	        //         IF #si_BinReleaseDistanceRight <= 0 THEN

	        //             #sx_Hold180 := TRUE;
	        //             #sx_ReleaseBinHoldRight := FALSE;
	        //             #sx_Hold170 := FALSE;
	        //             #sx_BinReleaseRight := FALSE;

	        //         END_IF;
	        //     END_IF;
	        // END_IF;

	    END_REGION


	    REGION Clearing sequence when workstation is deativated

	        #sF_TRIG_StationDeactivated(CLK := #ix_StationActive);



	        IF #sF_TRIG_StationDeactivated.Q THEN

	            #sx_Enable1X0In := TRUE;
	            #sx_Enable0X0In := TRUE;
	            #sx_Enable2X0In := TRUE;
	            #si_040DestinationA := 2;
	            #si_040DestinationB := 0;
	            #si_040DestinationC := 0;
	            #si_040DestinationD := 0;

	            #si_140DestinationA := 1;
	            #si_140DestinationB := 0;
	            #si_140DestinationC := 0;
	            #si_140DestinationD := 0;

	            #si_240DestinationA := 3;
	            #si_240DestinationB := 0;
	            #si_240DestinationC := 3;
	            #si_240DestinationD := 3;


	            #sx_Hold130 := FALSE;
	            #sx_Hold030 := FALSE;
	            #sx_Hold120 := FALSE;
	            #sx_Hold020 := FALSE;
	            #sx_Hold220 := FALSE;
	            #sx_Hold230 := FALSE;
	            #sx_Hold080 := FALSE;
	            #sx_Hold180 := FALSE;
	            #sx_StartClearing := TRUE;
	            #sx_NoOperationInProgress := FALSE;

	        END_IF;


	    END_REGION

	    REGION Finish operation

	        #sF_TRIG_ParcelArrived0X0(CLK := #iqUDT_WorkstationStatus."050".PEC_EoS.PEC);
	        #sF_TRIG_ParcelArrived1X0(CLK := #iqUDT_WorkstationStatus."150".PEC_EoS.PEC);
	        #sF_TRIG_ParcelArrived2X0(CLK := #iqUDT_WorkstationStatus."250".PEC_EoS.PEC);

	        // Check if operation if finished. If yes then set operation in progress bit
	        IF #si_SendTo0X0 AND #sF_TRIG_ParcelArrived0X0.Q OR #sFB_OperationTimeout.qx_DelayedSignal THEN

	            #si_SendTo0X0 := FALSE;

	        END_IF;


	        IF #si_SendTo1X0 AND #sF_TRIG_ParcelArrived1X0.Q OR #sFB_OperationTimeout.qx_DelayedSignal THEN

	            #si_SendTo1X0 := FALSE;

	        END_IF;

	        IF #si_SendTo2X0 AND #sF_TRIG_ParcelArrived2X0.Q OR #sFB_OperationTimeout.qx_DelayedSignal THEN

	            #si_SendTo2X0 := FALSE;

	        END_IF;


	        IF NOT #si_SendTo0X0 AND NOT #si_SendTo1X0 AND NOT #si_SendTo2X0 AND NOT #sx_StartClearing
	            AND #sUDT_Interface_040.ActualSpeed = 0
	            AND #sUDT_Interface_041.ActualSpeed = 0
	            AND #sUDT_Interface_140.ActualSpeed = 0
	            AND #sUDT_Interface_141.ActualSpeed = 0
	            AND #sUDT_Interface_240.ActualSpeed = 0
	            AND #sUDT_Interface_241.ActualSpeed = 0
	        THEN

	            #sx_NoOperationInProgress := TRUE;
	            #si_040DestinationA := 0;
	            #si_040DestinationB := 0;
	            #si_040DestinationC := 0;
	            #si_040DestinationD := 0;

	            #si_140DestinationA := 0;
	            #si_140DestinationB := 0;
	            #si_140DestinationC := 0;
	            #si_140DestinationD := 0;

	            #si_240DestinationA := 0;
	            #si_240DestinationB := 0;
	            #si_240DestinationC := 0;
	            #si_240DestinationD := 0;

	            #sx_Hold030 := FALSE;
	            #sx_Hold130 := FALSE;
	            #sx_Hold020 := FALSE;
	            #sx_Hold120 := FALSE;
	            #sx_Hold230 := FALSE;
	            #sx_Hold220 := FALSE;

	            #sx_Enable0X0In := FALSE;
	            #sx_Enable1X0In := FALSE;
	            #sx_Enable2X0In := FALSE;

	        END_IF;


	    END_REGION



	    REGION Workstation inicializaction

	        #sR_TRIG_InicializeWS(CLK := #ix_StationActive);

	        IF #sR_TRIG_InicializeWS.Q THEN

	            #sx_StartClearing := FALSE;
	            IF #iqUDT_WorkstationStatus."010".PEC_EoS.PEC THEN

	                #si_ReqestNewEmptyBin += 1;

	            END_IF;

	            IF #iqUDT_WorkstationStatus."020".PEC_EoS.PEC THEN

	                #si_ReqestNewEmptyBin += 1;

	            END_IF;

	            IF #iqUDT_WorkstationStatus."030".PEC_EoS.PEC THEN

	                #si_ReqestNewEmptyBin += 1;

	            END_IF;

	            IF #iqUDT_WorkstationStatus."110".PEC_EoS.PEC THEN

	                #si_ReqestNewPartialBin += 1;

	            END_IF;

	            IF #iqUDT_WorkstationStatus."120".PEC_EoS.PEC THEN

	                #si_ReqestNewPartialBin += 1;

	            END_IF;

	            IF #iqUDT_WorkstationStatus."130".PEC_EoS.PEC THEN

	                #si_ReqestNewPartialBin += 1;

	            END_IF;

	            #si_EmptyBinRequiredCounter0X0 := 2;
	            #si_EmptyBinRequiredCounter1X0 := 2;
	            #si_PartialyBinRequiredCounter0X0 := 1;
	            #si_PartialyBinRequiredCounter1X0 := 1;

	            REGION 050 Workposition inicialization
	                IF NOT #iqUDT_WorkstationStatus."050".PEC_EoS.PEC THEN
	                    IF #sa_TrackingArray_050[#iqUDT_Configuration."050".PEC_EoS.Distance / 10 - 2] > #iqUDT_Configuration.GlobalConfig.GINRangeStart
	                        AND #sa_TrackingArray_050[#iqUDT_Configuration."050".PEC_EoS.Distance / 10 - 2] < ((#iqUDT_Configuration.GlobalConfig.GINRangeStart + #iqUDT_Configuration.GlobalConfig.GINRangeEnd) / 2) THEN
	                        IF #si_EmptyBinRequiredCounter0X0 > 0 THEN
	                            #si_EmptyBinRequiredCounter0X0 -= 1;
	                        END_IF;
	                    ELSE

	                        IF #si_PartialyBinRequiredCounter0X0 > 0 THEN
	                            #si_PartialyBinRequiredCounter0X0 -= 1;
	                        ELSE
	                            IF #si_EmptyBinRequiredCounter0X0 > 0 THEN
	                                #si_EmptyBinRequiredCounter0X0 -= 1;
	                            END_IF;


	                        END_IF;

	                    END_IF;


	                END_IF;
	            END_REGION

	            REGION 060 Workposition inicialization
	                IF NOT #iqUDT_WorkstationStatus."060".PEC_EoS.PEC THEN
	                    IF #sa_TrackingArray_060[#iqUDT_Configuration."060".PEC_EoS.Distance / 10 - 2] > #iqUDT_Configuration.GlobalConfig.GINRangeStart
	                        AND #sa_TrackingArray_060[#iqUDT_Configuration."060".PEC_EoS.Distance / 10 - 2] < ((#iqUDT_Configuration.GlobalConfig.GINRangeStart + #iqUDT_Configuration.GlobalConfig.GINRangeEnd) / 2) THEN
	                        IF #si_EmptyBinRequiredCounter0X0 > 0 THEN
	                            #si_EmptyBinRequiredCounter0X0 -= 1;
	                        END_IF;
	                    ELSE

	                        IF #si_PartialyBinRequiredCounter0X0 > 0 THEN
	                            #si_PartialyBinRequiredCounter0X0 -= 1;
	                        ELSE
	                            IF #si_EmptyBinRequiredCounter0X0 > 0 THEN
	                                #si_EmptyBinRequiredCounter0X0 -= 1;
	                            END_IF;


	                        END_IF;

	                    END_IF;


	                END_IF;
	            END_REGION

	            REGION 070 Workposition inicialization
	                IF NOT #iqUDT_WorkstationStatus."070".PEC_EoS.PEC THEN
	                    IF #sa_TrackingArray_070[#iqUDT_Configuration."070".PEC_EoS.Distance / 10 - 2] > #iqUDT_Configuration.GlobalConfig.GINRangeStart
	                        AND #sa_TrackingArray_070[#iqUDT_Configuration."070".PEC_EoS.Distance / 10 - 2] < ((#iqUDT_Configuration.GlobalConfig.GINRangeStart + #iqUDT_Configuration.GlobalConfig.GINRangeEnd) / 2) THEN
	                        IF #si_EmptyBinRequiredCounter0X0 > 0 THEN
	                            #si_EmptyBinRequiredCounter0X0 -= 1;
	                        END_IF;
	                    ELSE

	                        IF #si_PartialyBinRequiredCounter0X0 > 0 THEN
	                            #si_PartialyBinRequiredCounter0X0 -= 1;
	                        ELSE
	                            IF #si_EmptyBinRequiredCounter0X0 > 0 THEN
	                                #si_EmptyBinRequiredCounter0X0 -= 1;
	                            END_IF;


	                        END_IF;

	                    END_IF;


	                END_IF;
	            END_REGION

	            REGION 150 Workposition inicialization
	                IF NOT #iqUDT_WorkstationStatus."150".PEC_EoS.PEC
	                THEN
	                    IF (#sa_TrackingArray_150[#iqUDT_Configuration."150".PEC_EoS.Distance / 10 / 10 - 2] > #iqUDT_Configuration.GlobalConfig.GINRangeStart
	                        AND #sa_TrackingArray_150[#iqUDT_Configuration."150".PEC_EoS.Distance / 10 - 2] < ((#iqUDT_Configuration.GlobalConfig.GINRangeStart + #iqUDT_Configuration.GlobalConfig.GINRangeEnd) / 2))
	                    THEN
	                        IF #si_EmptyBinRequiredCounter1X0 > 0 THEN
	                            #si_EmptyBinRequiredCounter1X0 -= 1;
	                        END_IF;
	                    ELSE

	                        IF #si_PartialyBinRequiredCounter1X0 > 0 THEN
	                            #si_PartialyBinRequiredCounter1X0 -= 1;
	                        ELSE
	                            IF #si_EmptyBinRequiredCounter1X0 > 0 THEN
	                                #si_EmptyBinRequiredCounter1X0 -= 1;
	                            END_IF;


	                        END_IF;

	                    END_IF;


	                END_IF;
	            END_REGION

	            REGION 160 Workposition inicialization
	                IF NOT #iqUDT_WorkstationStatus."160".PEC_EoS.PEC THEN
	                    IF #sa_TrackingArray_160[#iqUDT_Configuration."160".PEC_EoS.Distance / 10 - 2] > #iqUDT_Configuration.GlobalConfig.GINRangeStart
	                        AND #sa_TrackingArray_160[#iqUDT_Configuration."160".PEC_EoS.Distance / 10 - 2] < ((#iqUDT_Configuration.GlobalConfig.GINRangeStart + #iqUDT_Configuration.GlobalConfig.GINRangeEnd) / 2) THEN
	                        IF #si_EmptyBinRequiredCounter1X0 > 0 THEN
	                            #si_EmptyBinRequiredCounter1X0 -= 1;
	                        END_IF;
	                    ELSE

	                        IF #si_PartialyBinRequiredCounter1X0 > 0 THEN
	                            #si_PartialyBinRequiredCounter1X0 -= 1;
	                        ELSE
	                            IF #si_EmptyBinRequiredCounter1X0 > 0 THEN
	                                #si_EmptyBinRequiredCounter1X0 -= 1;
	                            END_IF;


	                        END_IF;

	                    END_IF;


	                END_IF;
	            END_REGION

	            REGION 170 Workposition inicialization
	                IF NOT #iqUDT_WorkstationStatus."170".PEC_EoS.PEC THEN
	                    IF #sa_TrackingArray_170[#iqUDT_Configuration."170".PEC_EoS.Distance / 10 - 2] > #iqUDT_Configuration.GlobalConfig.GINRangeStart
	                        AND #sa_TrackingArray_170[#iqUDT_Configuration."170".PEC_EoS.Distance / 10 - 2] < ((#iqUDT_Configuration.GlobalConfig.GINRangeStart + #iqUDT_Configuration.GlobalConfig.GINRangeEnd) / 2) THEN
	                        IF #si_EmptyBinRequiredCounter1X0 > 0 THEN
	                            #si_EmptyBinRequiredCounter1X0 -= 1;
	                        END_IF;
	                    ELSE

	                        IF #si_PartialyBinRequiredCounter1X0 > 0 THEN
	                            #si_PartialyBinRequiredCounter1X0 -= 1;
	                        ELSE
	                            IF #si_EmptyBinRequiredCounter1X0 > 0 THEN
	                                #si_EmptyBinRequiredCounter1X0 -= 1;
	                            END_IF;


	                        END_IF;

	                    END_IF;


	                END_IF;
	            END_REGION

	        END_IF;

	    END_REGION


	    REGION Request empty bin to buffer

	        IF #si_ReqestNewEmptyBin > 0 THEN

	            #ti_NumberOfBinInQueue := 0;
	            IF #iqUDT_EmptyBuffer.BufferState1.BinRequest THEN
	                #ti_NumberOfBinInQueue += 1;
	            END_IF;
	            IF #iqUDT_EmptyBuffer.BufferState2.BinRequest THEN
	                #ti_NumberOfBinInQueue += 1;
	            END_IF;
	            IF #iqUDT_EmptyBuffer.BufferState3.BinRequest THEN
	                #ti_NumberOfBinInQueue += 1;
	            END_IF;
	            IF NOT #iqUDT_WorkstationStatus."010".PEC_EoS.PEC THEN
	                #ti_NumberOfBinInQueue += 1;
	            END_IF;
	            IF NOT #iqUDT_WorkstationStatus."020".PEC_EoS.PEC THEN
	                #ti_NumberOfBinInQueue += 1;
	            END_IF;
	            IF NOT #iqUDT_WorkstationStatus."030".PEC_EoS.PEC THEN
	                #ti_NumberOfBinInQueue += 1;
	            END_IF;

	            IF #ti_NumberOfBinInQueue < 3 THEN

	                "FC_Fifo"(ic_Mode := 'S',
	                          qUDT_Status => #tUDT_FifoStatusEmpty,
	                          qx_Error => #tx_Error,
	                          qx_Warning => #tx_Warning,
	                          iqv_Data := #iqUDT_Configuration.GlobalConfig.DestinationEmpty,
	                          iqUDT_FifoHeader := #iqa_EmptyFifoHeader,
	                          iqv_DataBuffer := #iqa_EmptyFifoData);

	                IF NOT #tUDT_FifoStatusEmpty.FifoFull THEN

	                    "FC_Fifo"(ic_Mode := 'W',
	                              qUDT_Status => #tUDT_FifoStatusEmpty,
	                              qx_Error => #tx_Error,
	                              qx_Warning => #tx_Warning,
	                              iqv_Data := #iqUDT_Configuration.GlobalConfig.DestinationEmpty,
	                              iqUDT_FifoHeader := #iqa_EmptyFifoHeader,
	                              iqv_DataBuffer := #iqa_EmptyFifoData);

	                    IF NOT #iqUDT_EmptyBuffer.BufferState1.BinRequest THEN
	                        #iqUDT_EmptyBuffer.BufferState1.BinRequest := TRUE;
	                    ELSIF NOT #iqUDT_EmptyBuffer.BufferState2.BinRequest THEN
	                        #iqUDT_EmptyBuffer.BufferState2.BinRequest := TRUE;
	                    ELSE
	                        #iqUDT_EmptyBuffer.BufferState3.BinRequest := TRUE;
	                    END_IF;

	                    #si_ReqestNewEmptyBin -= 1;
	                    #iqUDT_EmptyBuffer.Destination := #iqUDT_Configuration.GlobalConfig.DestinationEmpty;
	                END_IF;



	            END_IF;

	        END_IF;


	    END_REGION

	    REGION Request partial bin to buffer

	        IF #si_ReqestNewPartialBin > 0 THEN

	            #ti_NumberOfBinInQueue := 0;
	            IF #iqUDT_PartialBuffer.BufferState1.BinRequest THEN
	                #ti_NumberOfBinInQueue += 1;
	            END_IF;
	            IF #iqUDT_PartialBuffer.BufferState2.BinRequest THEN
	                #ti_NumberOfBinInQueue += 1;
	            END_IF;
	            IF #iqUDT_PartialBuffer.BufferState3.BinRequest THEN
	                #ti_NumberOfBinInQueue += 1;
	            END_IF;
	            IF NOT #iqUDT_WorkstationStatus."110".PEC_EoS.PEC THEN
	                #ti_NumberOfBinInQueue += 1;
	            END_IF;
	            IF NOT #iqUDT_WorkstationStatus."120".PEC_EoS.PEC THEN
	                #ti_NumberOfBinInQueue += 1;
	            END_IF;
	            IF NOT #iqUDT_WorkstationStatus."130".PEC_EoS.PEC THEN
	                #ti_NumberOfBinInQueue += 1;
	            END_IF;

	            IF #ti_NumberOfBinInQueue < 3 THEN



	                "FC_Fifo"(ic_Mode := 'S',
	                          qUDT_Status => #tUDT_FifoStatusPartial,
	                          qx_Error => #tx_Error,
	                          qx_Warning => #tx_Warning,
	                          iqv_Data := #iqUDT_Configuration.GlobalConfig.DestinationPartialy,
	                          iqUDT_FifoHeader := #iqa_PartialFifoHeader,
	                          iqv_DataBuffer := #iqa_PartialFifoData);

	                IF NOT #tUDT_FifoStatusPartial.FifoFull THEN

	                    "FC_Fifo"(ic_Mode := 'W',
	                              qUDT_Status => #tUDT_FifoStatusPartial,
	                              qx_Error => #tx_Error,
	                              qx_Warning => #tx_Warning,
	                              iqv_Data := #iqUDT_Configuration.GlobalConfig.DestinationPartialy,
	                              iqUDT_FifoHeader := #iqa_PartialFifoHeader,
	                              iqv_DataBuffer := #iqa_PartialFifoData);

	                    IF NOT #iqUDT_PartialBuffer.BufferState1.BinRequest THEN
	                        #iqUDT_PartialBuffer.BufferState1.BinRequest := TRUE;
	                    ELSIF NOT #iqUDT_PartialBuffer.BufferState2.BinRequest THEN
	                        #iqUDT_PartialBuffer.BufferState2.BinRequest := TRUE;
	                    ELSE
	                        #iqUDT_PartialBuffer.BufferState3.BinRequest := TRUE;
	                    END_IF;

	                    #si_ReqestNewPartialBin -= 1;
	                    #iqUDT_PartialBuffer.Destination := #iqUDT_Configuration.GlobalConfig.DestinationPartialy;

	                END_IF;

	            END_IF;

	        END_IF;

	    END_REGION

	    REGION Ordered bin monitoring

	        IF "DB_Memory".OS_2sec THEN

	            IF #iqUDT_EmptyBuffer.BufferState1.BinSend THEN
	                #iqUDT_EmptyBuffer.BufferState1.WaintingTime += 2;

	                IF #iqUDT_EmptyBuffer.BufferState1.WaintingTime > #iqUDT_Configuration.GlobalConfig.BinOrderTimeout THEN

	                    #iqUDT_EmptyBuffer.BufferState1 := #iqUDT_EmptyBuffer.BufferState2;
	                    #iqUDT_EmptyBuffer.BufferState2 := #iqUDT_EmptyBuffer.BufferState3;

	                    #iqUDT_EmptyBuffer.BufferState3.BinSend := FALSE;
	                    #iqUDT_EmptyBuffer.BufferState3.BinRequest := FALSE;
	                    #iqUDT_EmptyBuffer.BufferState3.UpcomingBarcode := '';
	                    #iqUDT_EmptyBuffer.BufferState3.WaintingTime := 0;


	                    #ti_NumberOfBinInQueue := 0;
	                    IF #iqUDT_EmptyBuffer.BufferState1.BinRequest THEN
	                        #ti_NumberOfBinInQueue += 1;
	                    END_IF;
	                    IF #iqUDT_EmptyBuffer.BufferState2.BinRequest THEN
	                        #ti_NumberOfBinInQueue += 1;
	                    END_IF;
	                    IF NOT #iqUDT_WorkstationStatus."010".PEC_EoS.PEC THEN
	                        #ti_NumberOfBinInQueue += 1;
	                    END_IF;
	                    IF NOT #iqUDT_WorkstationStatus."020".PEC_EoS.PEC THEN
	                        #ti_NumberOfBinInQueue += 1;
	                    END_IF;
	                    IF NOT #iqUDT_WorkstationStatus."030".PEC_EoS.PEC THEN
	                        #ti_NumberOfBinInQueue += 1;
	                    END_IF;

	                    IF #ti_NumberOfBinInQueue < 3 THEN
	                        #si_ReqestNewEmptyBin += 1;
	                    END_IF;


	                END_IF;

	            END_IF;

	            IF #iqUDT_EmptyBuffer.BufferState2.BinSend THEN
	                #iqUDT_EmptyBuffer.BufferState2.WaintingTime += 2;

	                IF #iqUDT_EmptyBuffer.BufferState2.WaintingTime > #iqUDT_Configuration.GlobalConfig.BinOrderTimeout THEN

	                    #iqUDT_EmptyBuffer.BufferState2 := #iqUDT_EmptyBuffer.BufferState3;

	                    #iqUDT_EmptyBuffer.BufferState3.BinSend := FALSE;
	                    #iqUDT_EmptyBuffer.BufferState3.BinRequest := FALSE;
	                    #iqUDT_EmptyBuffer.BufferState3.UpcomingBarcode := '';
	                    #iqUDT_EmptyBuffer.BufferState3.WaintingTime := 0;

	                    #si_ReqestNewEmptyBin += 1;

	                END_IF;

	            END_IF;

	            IF #iqUDT_EmptyBuffer.BufferState3.BinSend THEN
	                #iqUDT_EmptyBuffer.BufferState3.WaintingTime += 2;

	                IF #iqUDT_EmptyBuffer.BufferState3.WaintingTime > #iqUDT_Configuration.GlobalConfig.BinOrderTimeout THEN

	                    #iqUDT_EmptyBuffer.BufferState3.BinSend := FALSE;
	                    #iqUDT_EmptyBuffer.BufferState3.BinRequest := FALSE;
	                    #iqUDT_EmptyBuffer.BufferState3.UpcomingBarcode := '';
	                    #iqUDT_EmptyBuffer.BufferState3.WaintingTime := 0;
	                    #si_ReqestNewEmptyBin += 1;

	                END_IF;

	            END_IF;

	            IF #iqUDT_PartialBuffer.BufferState1.BinSend THEN
	                #iqUDT_PartialBuffer.BufferState1.WaintingTime += 2;

	                IF #iqUDT_PartialBuffer.BufferState1.WaintingTime > #iqUDT_Configuration.GlobalConfig.BinOrderTimeout THEN

	                    #iqUDT_PartialBuffer.BufferState1 := #iqUDT_PartialBuffer.BufferState2;
	                    #iqUDT_PartialBuffer.BufferState2 := #iqUDT_PartialBuffer.BufferState3;
	                    #iqUDT_PartialBuffer.BufferState3.BinSend := FALSE;
	                    #iqUDT_PartialBuffer.BufferState3.BinRequest := FALSE;
	                    #iqUDT_PartialBuffer.BufferState3.UpcomingBarcode := '';
	                    #iqUDT_PartialBuffer.BufferState3.WaintingTime := 0;


	                    #ti_NumberOfBinInQueue := 0;
	                    IF #iqUDT_PartialBuffer.BufferState1.BinRequest THEN
	                        #ti_NumberOfBinInQueue += 1;
	                    END_IF;
	                    IF #iqUDT_PartialBuffer.BufferState2.BinRequest THEN
	                        #ti_NumberOfBinInQueue += 1;
	                    END_IF;
	                    IF NOT #iqUDT_WorkstationStatus."110".PEC_EoS.PEC THEN
	                        #ti_NumberOfBinInQueue += 1;
	                    END_IF;
	                    IF NOT #iqUDT_WorkstationStatus."120".PEC_EoS.PEC THEN
	                        #ti_NumberOfBinInQueue += 1;
	                    END_IF;
	                    IF NOT #iqUDT_WorkstationStatus."130".PEC_EoS.PEC THEN
	                        #ti_NumberOfBinInQueue += 1;
	                    END_IF;

	                    IF #ti_NumberOfBinInQueue < 3 THEN
	                        #si_ReqestNewPartialBin += 1;
	                    END_IF;

	                END_IF;

	            END_IF;


	            IF #iqUDT_PartialBuffer.BufferState2.BinSend THEN
	                #iqUDT_PartialBuffer.BufferState2.WaintingTime += 2;
	                IF #iqUDT_PartialBuffer.BufferState2.WaintingTime > #iqUDT_Configuration.GlobalConfig.BinOrderTimeout THEN

	                    #iqUDT_PartialBuffer.BufferState2 := #iqUDT_PartialBuffer.BufferState3;

	                    #iqUDT_PartialBuffer.BufferState3.BinSend := FALSE;
	                    #iqUDT_PartialBuffer.BufferState3.BinRequest := FALSE;
	                    #iqUDT_PartialBuffer.BufferState3.UpcomingBarcode := '';
	                    #iqUDT_PartialBuffer.BufferState3.WaintingTime := 0;

	                    #si_ReqestNewPartialBin += 1;

	                END_IF;

	            END_IF;

	            IF #iqUDT_PartialBuffer.BufferState3.BinSend THEN
	                #iqUDT_PartialBuffer.BufferState3.WaintingTime += 2;

	                IF #iqUDT_PartialBuffer.BufferState3.WaintingTime > #iqUDT_Configuration.GlobalConfig.BinOrderTimeout THEN

	                    #iqUDT_PartialBuffer.BufferState3.BinSend := FALSE;
	                    #iqUDT_PartialBuffer.BufferState3.BinRequest := FALSE;
	                    #iqUDT_PartialBuffer.BufferState3.UpcomingBarcode := '';
	                    #iqUDT_PartialBuffer.BufferState3.WaintingTime := 0;
	                    #si_ReqestNewPartialBin += 1;

	                END_IF;
	            END_IF;

	        END_IF;

	    END_REGION

	    REGION Ordered product confirmation

	        REGION Empty

	            #sR_TRIG_EmptyBinReceived(CLK := #sa_TrackingArray_010[#iqUDT_Configuration."010".PEC_EoS.Distance / 10 - 1] <> 0);

	            IF #sR_TRIG_EmptyBinReceived.Q THEN

	                IF #iqUDT_EmptyBuffer.BufferState1.BinSend AND "DB_GIN".GIN[#sa_TrackingArray_010[#iqUDT_Configuration."010".PEC_EoS.Distance / 10 - 1]].WES.Barcode = #iqUDT_EmptyBuffer.BufferState1.UpcomingBarcode THEN

	                    #iqUDT_EmptyBuffer.BufferState1 := #iqUDT_EmptyBuffer.BufferState2;
	                    #iqUDT_EmptyBuffer.BufferState2 := #iqUDT_EmptyBuffer.BufferState3;

	                    #iqUDT_EmptyBuffer.BufferState3.BinSend := FALSE;
	                    #iqUDT_EmptyBuffer.BufferState3.BinRequest := FALSE;
	                    #iqUDT_EmptyBuffer.BufferState3.UpcomingBarcode := '';
	                    #iqUDT_EmptyBuffer.BufferState3.WaintingTime := 0;
	                END_IF;


	                IF #iqUDT_EmptyBuffer.BufferState2.BinSend AND "DB_GIN".GIN[#sa_TrackingArray_010[#iqUDT_Configuration."010".PEC_EoS.Distance / 10 - 1]].WES.Barcode = #iqUDT_EmptyBuffer.BufferState2.UpcomingBarcode THEN

	                    #iqUDT_EmptyBuffer.BufferState2 := #iqUDT_EmptyBuffer.BufferState3;

	                    #iqUDT_EmptyBuffer.BufferState3.BinSend := FALSE;
	                    #iqUDT_EmptyBuffer.BufferState3.BinRequest := FALSE;
	                    #iqUDT_EmptyBuffer.BufferState3.UpcomingBarcode := '';
	                    #iqUDT_EmptyBuffer.BufferState3.WaintingTime := 0;
	                END_IF;


	                IF #iqUDT_EmptyBuffer.BufferState3.BinSend AND "DB_GIN".GIN[#sa_TrackingArray_010[#iqUDT_Configuration."010".PEC_EoS.Distance / 10 - 1]].WES.Barcode = #iqUDT_EmptyBuffer.BufferState3.UpcomingBarcode THEN

	                    #iqUDT_EmptyBuffer.BufferState3.BinSend := FALSE;
	                    #iqUDT_EmptyBuffer.BufferState3.BinRequest := FALSE;
	                    #iqUDT_EmptyBuffer.BufferState3.UpcomingBarcode := '';
	                    #iqUDT_EmptyBuffer.BufferState3.WaintingTime := 0;
	                END_IF;

	            END_IF;

	        END_REGION

	        REGION Partialy


	            #sR_TRIG_PartialBinReceived(CLK := #sa_TrackingArray_110[#iqUDT_Configuration."110".PEC_EoS.Distance / 10 - 1] <> 0);

	            IF #sR_TRIG_PartialBinReceived.Q THEN

	                IF #iqUDT_PartialBuffer.BufferState1.BinSend AND "DB_GIN".GIN[#sa_TrackingArray_110[#iqUDT_Configuration."110".PEC_EoS.Distance / 10 - 1]].WES.Barcode = #iqUDT_PartialBuffer.BufferState1.UpcomingBarcode THEN

	                    #iqUDT_PartialBuffer.BufferState1 := #iqUDT_PartialBuffer.BufferState2;
	                    #iqUDT_PartialBuffer.BufferState2 := #iqUDT_PartialBuffer.BufferState3;

	                    #iqUDT_PartialBuffer.BufferState3.BinSend := FALSE;
	                    #iqUDT_PartialBuffer.BufferState3.BinRequest := FALSE;
	                    #iqUDT_PartialBuffer.BufferState3.UpcomingBarcode := '';
	                    #iqUDT_PartialBuffer.BufferState3.WaintingTime := 0;
	                END_IF;


	                IF #iqUDT_PartialBuffer.BufferState2.BinSend AND "DB_GIN".GIN[#sa_TrackingArray_110[#iqUDT_Configuration."110".PEC_EoS.Distance / 10 - 1]].WES.Barcode = #iqUDT_PartialBuffer.BufferState2.UpcomingBarcode THEN

	                    #iqUDT_PartialBuffer.BufferState2 := #iqUDT_PartialBuffer.BufferState3;

	                    #iqUDT_PartialBuffer.BufferState3.BinSend := FALSE;
	                    #iqUDT_PartialBuffer.BufferState3.BinRequest := FALSE;
	                    #iqUDT_PartialBuffer.BufferState3.UpcomingBarcode := '';
	                    #iqUDT_PartialBuffer.BufferState3.WaintingTime := 0;
	                END_IF;


	                IF #iqUDT_PartialBuffer.BufferState3.BinSend AND "DB_GIN".GIN[#sa_TrackingArray_110[#iqUDT_Configuration."110".PEC_EoS.Distance / 10 - 1]].WES.Barcode = #iqUDT_PartialBuffer.BufferState3.UpcomingBarcode THEN

	                    #iqUDT_PartialBuffer.BufferState3.BinSend := FALSE;
	                    #iqUDT_PartialBuffer.BufferState3.BinRequest := FALSE;
	                    #iqUDT_PartialBuffer.BufferState3.UpcomingBarcode := '';
	                    #iqUDT_PartialBuffer.BufferState3.WaintingTime := 0;
	                END_IF;

	            END_IF;

	        END_REGION


	    END_REGION

	END_REGION

	REGION 010

	    REGION Change GIN range

	        #sR_TRIG_NewParcel010(CLK := #iqUDT_HandshakeUpstream010.GIN <> 0);

	        IF #sR_TRIG_NewParcel010.Q THEN

	            #si_LastGIN010 += 1;

	            IF #si_LastGIN010 < #iqUDT_Configuration.GlobalConfig.GINRangeStart
	                OR #si_LastGIN010 > ((#iqUDT_Configuration.GlobalConfig.GINRangeStart + #iqUDT_Configuration.GlobalConfig.GINRangeEnd) / 2)
	            THEN
	                #si_LastGIN010 := #iqUDT_Configuration.GlobalConfig.GINRangeStart;
	            END_IF;
	            #ts_Barcode := "DB_GIN".GIN[#iqUDT_HandshakeUpstream010.GIN].WES.Barcode;
	            #iqUDT_HandshakeUpstream010.GIN := #si_LastGIN010;
	            "DB_GIN".GIN[#iqUDT_HandshakeUpstream010.GIN] := "DB_GINDefault".GIN[#iqUDT_Configuration."010".PEC_EoS.DefaultGIN];
	            "DB_GIN".GIN[#iqUDT_HandshakeUpstream010.GIN].WES.Barcode := #ts_Barcode;
	        END_IF;

	    END_REGION

	    REGION Displacement
	        #sFB_Displacement010(#sUDT_Interface_010);
	    END_REGION

	    REGION Tracking

	        #sFB_Tracking_010(iUDT_ConveyorCommonConfiguration := #iqUDT_Configuration."010".Conveyor.Common,
	                          iqa_TrackingData := #sa_TrackingArray_010,
	                          iqUDT_ConveyorInterface := #sUDT_Interface_010,
	                          iqUDT_HandshakeUp := #iqUDT_HandshakeUpstream010,
	                          iqUDT_Handshake := #sUDT_Handshake_010);

	    END_REGION

	    REGION EoS

	        #sFB_PECUpdate_010(iUDT_PECUpdateConfiguration := #iqUDT_Configuration."010".PEC_EoS,
	                           iUDT_ConveyorCommonConfiguration := #iqUDT_Configuration."010".Conveyor.Common,
	                           ix_PEC := #iUDT_MotorInput010.AllSensorPortInputs.LeftSensor,
	                           ix_TeachingMode := FALSE,
	                           qUDT_Status => #iqUDT_WorkstationStatus."010".PEC_EoS,
	                           iqUDT_ConveyorInterface := #sUDT_Interface_010,
	                           iqUDT_UnknownGINRange := #iqUDT_UnknownGINRange,
	                           iqUDT_FifoHeader := "DB_FIFOLostGIN".Header,
	                           iqUDT_Statistics := #iqUDT_WorkstationStatistics."010".PEC_EoS,
	                           iqa_TrackingData := #sa_TrackingArray_010,
	                           iqa_FifoData := "DB_FIFOLostGIN".Data);

	    END_REGION

	    REGION Conveyor

	        #sFB_Conveyor_010(iUDT_ConveyorConfiguration := #iqUDT_Configuration."010".Conveyor,
	                          idi_PECEoSDistance := #iqUDT_Configuration."010".PEC_EoS.Distance,
	                          idi_PECBoSDistance := 0,
	                          ii_ExternalSpeed := 0,
	                          ix_SafetyOk := #ix_SafetyOk,
	                          ix_24vOk := #ix_24vOk,
	                          ix_400vOk := #ix_400vOk,
	                          ix_HardwareOk := TRUE,
	                          ix_PECEoS := #iqUDT_WorkstationStatus."010".PEC_EoS.PEC,
	                          ix_PECBoS := TRUE,
	                          ix_ReverseDirection := FALSE,
	                          ix_ExternalRequestDieBack := (#sUDT_Interface_020.ActualSpeed = 0 AND NOT #iqUDT_WorkstationStatus."010".PEC_EoS.PEC),
	                          ix_ExternalRequestHold := FALSE,
	                          ix_ResetEnergySave := FALSE,
	                          qUDT_HMIStatus => #iqUDT_WorkstationStatus."010".Conveyor,
	                          qUDT_Status => #iqUDT_WorkstationCommonStatus."010",
	                          iqUDT_EquipmentControl := #iqUDT_EquipmentControl,
	                          iqUDT_ConveyorCommand := #iqUDT_WorkstationCommands."010".Conveyor,
	                          iqUDT_ConveyorInterface := #sUDT_Interface_010,
	                          iqUDT_HandShakeUp := #iqUDT_HandshakeUpstream010,
	                          iqUDT_HandShake := #sUDT_Handshake_010,
	                          iqUDT_Statistics := #iqUDT_WorkstationStatistics."010".Conveyor);

	        // #iqUDT_HandshakeUpstream010.RTR := #iqUDT_HandshakeUpstream010.RTR AND #iqUDT_WorkstationStatus."010".PEC_EoS.PEC;

	    END_REGION

	    REGION MCO

	        #sFB_MCOConveyLinxAixController_010(iUDT_AixConfig := #iqUDT_Configuration."010".MCO_M01,
	                                            iUDT_AixInputsModule := #iUDT_MotorInput010,
	                                            ix_24vOk := #ix_24vOk,
	                                            ix_SimulationModeActive := "DB_Memory".Simulation,
	                                            ii_MotorPositionId := 1,
	                                            qUDT_HMIStatus => #iqUDT_WorkstationStatus."010".MCO_M01,
	                                            iqUDT_AixOutputsModule := #iqUDT_MotorOutput010,
	                                            iqUDT_ConveyorInterface := #sUDT_Interface_010,
	                                            iqUDT_MCOStatistics := #iqUDT_WorkstationStatistics."010".MCO_M01);
	    END_REGION

	END_REGION

	REGION 020

	    REGION Displacement
	        #sFB_Displacement020(#sUDT_Interface_020);
	    END_REGION

	    REGION Tracking

	        #sFB_Tracking_020(iUDT_ConveyorCommonConfiguration := #iqUDT_Configuration."020".Conveyor.Common,
	                          iqa_TrackingData := #sa_TrackingArray_020,
	                          iqUDT_ConveyorInterface := #sUDT_Interface_020,
	                          iqUDT_HandshakeUp := #sUDT_Handshake_010,
	                          iqUDT_Handshake := #sUDT_Handshake_020);

	    END_REGION

	    REGION EoS

	        #sFB_PECUpdate_020(iUDT_PECUpdateConfiguration := #iqUDT_Configuration."020".PEC_EoS,
	                           iUDT_ConveyorCommonConfiguration := #iqUDT_Configuration."020".Conveyor.Common,
	                           ix_PEC := #iUDT_MotorInput010.AllSensorPortInputs.RightSensor,
	                           ix_TeachingMode := FALSE,
	                           qUDT_Status => #iqUDT_WorkstationStatus."020".PEC_EoS,
	                           iqUDT_ConveyorInterface := #sUDT_Interface_020,
	                           iqUDT_UnknownGINRange := #iqUDT_UnknownGINRange,
	                           iqUDT_FifoHeader := "DB_FIFOLostGIN".Header,
	                           iqUDT_Statistics := #iqUDT_WorkstationStatistics."020".PEC_EoS,
	                           iqa_TrackingData := #sa_TrackingArray_020,
	                           iqa_FifoData := "DB_FIFOLostGIN".Data);




	    END_REGION

	    REGION Conveyor

	        #sFB_Conveyor_020(iUDT_ConveyorConfiguration := #iqUDT_Configuration."020".Conveyor,
	                          idi_PECEoSDistance := #iqUDT_Configuration."020".PEC_EoS.Distance,
	                          idi_PECBoSDistance := 0,
	                          ii_ExternalSpeed := 0,
	                          ix_SafetyOk := #ix_SafetyOk,
	                          ix_24vOk := #ix_24vOk,
	                          ix_400vOk := #ix_400vOk,
	                          ix_HardwareOk := TRUE,
	                          ix_PECEoS := #iqUDT_WorkstationStatus."020".PEC_EoS.PEC,
	                          ix_PECBoS := TRUE,
	                          ix_ReverseDirection := FALSE,
	                          ix_ExternalRequestDieBack := #sx_Hold020 OR (#sUDT_Interface_030.ActualSpeed = 0 AND NOT #iqUDT_WorkstationStatus."020".PEC_EoS.PEC),
	                          ix_ExternalRequestHold := FALSE,
	                          ix_ResetEnergySave := FALSE,
	                          qUDT_HMIStatus => #iqUDT_WorkstationStatus."020".Conveyor,
	                          qUDT_Status => #iqUDT_WorkstationCommonStatus."020",
	                          iqUDT_EquipmentControl := #iqUDT_EquipmentControl,
	                          iqUDT_ConveyorCommand := #iqUDT_WorkstationCommands."020".Conveyor,
	                          iqUDT_ConveyorInterface := #sUDT_Interface_020,
	                          iqUDT_HandShakeUp := #sUDT_Handshake_010,
	                          iqUDT_HandShake := #sUDT_Handshake_020,
	                          iqUDT_Statistics := #iqUDT_WorkstationStatistics."020".Conveyor);

	    END_REGION

	    REGION MCO

	        #sFB_MCOConveyLinxAixController_020(iUDT_AixConfig := #iqUDT_Configuration."020".MCO_M01,
	                                            iUDT_AixInputsModule := #iUDT_MotorInput010,
	                                            ix_24vOk := #ix_24vOk,
	                                            ix_SimulationModeActive := "DB_Memory".Simulation,
	                                            ii_MotorPositionId := 2,
	                                            qUDT_HMIStatus => #iqUDT_WorkstationStatus."020".MCO_M01,
	                                            iqUDT_AixOutputsModule := #iqUDT_MotorOutput010,
	                                            iqUDT_ConveyorInterface := #sUDT_Interface_020,
	                                            iqUDT_MCOStatistics := #iqUDT_WorkstationStatistics."020".MCO_M01);
	    END_REGION

	END_REGION

	REGION 030

	    REGION Displacement
	        #sFB_Displacement030(#sUDT_Interface_030);
	    END_REGION

	    REGION Tracking

	        #sFB_Tracking_030(iUDT_ConveyorCommonConfiguration := #iqUDT_Configuration."030".Conveyor.Common,
	                          iqa_TrackingData := #sa_TrackingArray_030,
	                          iqUDT_ConveyorInterface := #sUDT_Interface_030,
	                          iqUDT_HandshakeUp := #sUDT_Handshake_020,
	                          iqUDT_Handshake := #sUDT_Handshake_030);

	    END_REGION

	    REGION EoS

	        #sFB_PECUpdate_030(iUDT_PECUpdateConfiguration := #iqUDT_Configuration."030".PEC_EoS,
	                           iUDT_ConveyorCommonConfiguration := #iqUDT_Configuration."030".Conveyor.Common,
	                           ix_PEC := #iUDT_MotorInput030.AllSensorPortInputs.LeftSensor,
	                           ix_TeachingMode := FALSE,
	                           qUDT_Status => #iqUDT_WorkstationStatus."030".PEC_EoS,
	                           iqUDT_ConveyorInterface := #sUDT_Interface_030,
	                           iqUDT_UnknownGINRange := #iqUDT_UnknownGINRange,
	                           iqUDT_FifoHeader := "DB_FIFOLostGIN".Header,
	                           iqUDT_Statistics := #iqUDT_WorkstationStatistics."030".PEC_EoS,
	                           iqa_TrackingData := #sa_TrackingArray_030,
	                           iqa_FifoData := "DB_FIFOLostGIN".Data);




	    END_REGION

	    REGION Conveyor

	        #sUDT_Handshake_030.RTR := #sUDT_Handshake_030.RTR AND NOT #sx_Hold030 OR #iqUDT_WorkstationStatus."030".PEC_EoS.PEC;


	        #sFB_Conveyor_030(iUDT_ConveyorConfiguration := #iqUDT_Configuration."030".Conveyor,
	                          idi_PECEoSDistance := #iqUDT_Configuration."030".PEC_EoS.Distance,
	                          idi_PECBoSDistance := 0,
	                          ii_ExternalSpeed := 0,
	                          ix_SafetyOk := #ix_SafetyOk,
	                          ix_24vOk := #ix_24vOk,
	                          ix_400vOk := #ix_400vOk,
	                          ix_HardwareOk := TRUE,
	                          ix_PECEoS := #iqUDT_WorkstationStatus."030".PEC_EoS.PEC,
	                          ix_PECBoS := TRUE,
	                          ix_ReverseDirection := FALSE,
	                          ix_ExternalRequestDieBack := FALSE,
	                          ix_ExternalRequestHold := #sx_Hold030,
	                          ix_ResetEnergySave := FALSE,
	                          qUDT_HMIStatus => #iqUDT_WorkstationStatus."030".Conveyor,
	                          qUDT_Status => #iqUDT_WorkstationCommonStatus."030",
	                          iqUDT_EquipmentControl := #iqUDT_EquipmentControl,
	                          iqUDT_ConveyorCommand := #iqUDT_WorkstationCommands."030".Conveyor,
	                          iqUDT_ConveyorInterface := #sUDT_Interface_030,
	                          iqUDT_HandShakeUp := #sUDT_Handshake_020,
	                          iqUDT_HandShake := #sUDT_Handshake_030,
	                          iqUDT_Statistics := #iqUDT_WorkstationStatistics."030".Conveyor);

	    END_REGION

	    REGION MCO

	        #sFB_MCOConveyLinxAixController_030(iUDT_AixConfig := #iqUDT_Configuration."030".MCO_M01,
	                                            iUDT_AixInputsModule := #iUDT_MotorInput030,
	                                            ix_24vOk := #ix_24vOk,
	                                            ix_SimulationModeActive := "DB_Memory".Simulation,
	                                            ii_MotorPositionId := 1,
	                                            qUDT_HMIStatus => #iqUDT_WorkstationStatus."030".MCO_M01,
	                                            iqUDT_AixOutputsModule := #iqUDT_MotorOutput030,
	                                            iqUDT_ConveyorInterface := #sUDT_Interface_030,
	                                            iqUDT_MCOStatistics := #iqUDT_WorkstationStatistics."030".MCO_M01);
	    END_REGION

	END_REGION

	REGION 040

	    REGION Displacement
	        #sFB_Displacement040(#sUDT_Interface_040);
	    END_REGION

	    REGION MCO

	        #sFB_MCOConveyLinxAixController_040(iUDT_AixConfig := #iqUDT_Configuration."040".MCO_M01,
	                                            iUDT_AixInputsModule := #iUDT_MotorInput040,
	                                            ii_PositionSetpoint := #iqUDT_RATPositioning040.Lower.EndPosition,
	                                            ix_24vOk := #ix_24vOk,
	                                            ix_SimulationModeActive := "DB_Memory".Simulation,
	                                            ii_MotorPositionId := 1,
	                                            ix_StartPositioning := #iqUDT_RATPositioning040.Lower.Start,
	                                            ix_ResetPosition := #iqUDT_RATPositioning040.Lower.ResetPosition,
	                                            qUDT_HMIStatus => #iqUDT_WorkstationStatus."040".MCO_M01,
	                                            qx_Positioned => #iqUDT_RATPositioning040.Lower.Done,
	                                            iqUDT_AixOutputsModule := #iqUDT_MotorOutput040,
	                                            iqUDT_ConveyorInterface := #sUDT_Interface_040,
	                                            iqUDT_MCOStatistics := #iqUDT_WorkstationStatistics."040".MCO_M01);
	    END_REGION

	    REGION BladeStopEoS

	        IF #iqUDT_Configuration.GlobalConfig.LeftStationAvailable THEN

	            #sFB_BladeStopEoS_040(iUDT_Configuration := #iqUDT_Configuration."040".BladeStopEoS,
	                                  ix_IsOpened := #ix_BladeStopisUp040,
	                                  ix_IsClosed := #ix_BladeStopisDown040,
	                                  ix_AirPressureOk := TRUE,
	                                  qx_Open => #qx_BladeStopControl040,
	                                  qUDT_HMIStatus => #iqUDT_WorkstationStatus."040".BladeStopEoS,
	                                  qUDT_Statistics => #iqUDT_WorkstationStatistics."040".BladeStopEoS,
	                                  iqUDT_EquipmentControl := #iqUDT_EquipmentControl,
	                                  iqUDT_HMICommand := #iqUDT_WorkstationCommands."040".BladeStopEoS,
	                                  iqUDT_Interface := #sUDT_Interface_040_BladeStopEoS);
	        END_IF;

	    END_REGION

	END_REGION

	REGION 041

	    REGION Displacement
	        #sFB_Displacement041(#sUDT_Interface_041);
	    END_REGION

	    REGION RAT

	        #iqUDT_Configuration."041".RightAngledTransfer.BladeStopEoS := #iqUDT_Configuration.GlobalConfig.LeftStationAvailable;

	        #sFB_RightAngledTransfer_041(iUDT_Configuration := #iqUDT_Configuration."041".RightAngledTransfer,
	                                     iUDT_LowerConveyorConfiguration := #iqUDT_Configuration."040".Conveyor,
	                                     iUDT_UpperConveyorConfiguration := #iqUDT_Configuration."041".Conveyor,
	                                     iUDT_PECConfiguration := #iqUDT_Configuration."040".PEC_EoS,
	                                     ii_DestinationA := #si_040DestinationA,
	                                     ii_DestinationB := #si_040DestinationB,
	                                     ii_DestinationC := #si_040DestinationC,
	                                     ii_DestinationD := #si_040DestinationD,
	                                     ix_HardwareOk := TRUE,
	                                     ix_400vOk := #ix_400vOk,
	                                     ix_24vOk := #ix_24vOk,
	                                     ix_SafetyOk := #ix_SafetyOk,
	                                     ix_AirPressureOk := #ix_AirPressureOk,
	                                     ix_SectionIsDown := #ix_SectionisDown041,
	                                     ix_SectionIsUp := #ix_SectionisUp041,
	                                     ix_ConveyorAAuto := #iqUDT_WorkstationCommonStatus."030".AutoON,
	                                     ix_ConveyorBAuto := #iqUDT_WorkstationCommonStatus."050".AutoON,
	                                     ix_ConveyorCAuto := FALSE,
	                                     ix_ConveyorDAuto := #iqUDT_WorkstationCommonStatus."241".AutoON,
	                                     ix_PEC := #iUDT_MotorInput040.AllSensorPortInputs.LeftSensor,
	                                     ix_ExternalReceiveRequestA := NOT #iqUDT_WorkstationStatus."030".PEC_EoS.PEC AND #sx_Enable0X0In,
	                                     ix_ExternalReceiveRequestB := false,
	                                     ix_ExternalReceiveRequestC := false,
	                                     ix_ExternalReceiveRequestD := #sFB_RightAngledTransfer_241.qx_ExternalSendRequestD,
	                                     ix_PECInfeedA := #iqUDT_WorkstationStatus."030".PEC_EoS.PEC,
	                                     ix_PECInfeedD := #iqUDT_WorkstationStatus."240".PEC_EoS.PEC,
	                                     qUDT_HMIRATStatus => #iqUDT_WorkstationStatus."041".RightAngledTransfer,
	                                     qUDT_HMIConveyorStatus => #iqUDT_WorkstationStatus."040".Conveyor,
	                                     qUDT_HMIPECStatus => #iqUDT_WorkstationStatus."040".PEC_EoS,
	                                     qUDT_RATStatus => #iqUDT_WorkstationCommonStatus."041",
	                                     qUDT_ConveyorStatus => #iqUDT_WorkstationCommonStatus."040",
	                                     qx_PopupControl => #qx_PopupControl041,
	                                     iqUDT_EquipmentControl := #iqUDT_EquipmentControl,
	                                     iqUDT_RATCommand := #iqUDT_WorkstationCommands."041".RightAngledTransfer,
	                                     iqUDT_ConveyorCommand := #iqUDT_WorkstationCommands."040".Conveyor,
	                                     iqUDT_RATStatistics := #iqUDT_WorkstationStatistics."041".RightAngledTransfer,
	                                     iqUDT_ConveyorStatistics := #iqUDT_WorkstationStatistics."040".Conveyor,
	                                     iqUDT_PECStatistics := #iqUDT_WorkstationStatistics."040".PEC_EoS,
	                                     iqUDT_HandShakeConveyorA := #sUDT_Handshake_030,
	                                     iqUDT_HandShakeConveyorB := #sUDT_Handshake_040,
	                                     iqUDT_HandShakeConveyorC := #sUDT_HandshakeUp_041,
	                                     iqUDT_HandShakeConveyorD := #sUDT_Handshake_041,
	                                     iqUDT_LowerConveyorInterface := #sUDT_Interface_040,
	                                     iqUDT_UpperConveyorInterface := #sUDT_Interface_041,
	                                     iqUDT_RATPositioning := #iqUDT_RATPositioning040,
	                                     iqUDT_BladeStopEoSInterface := #sUDT_Interface_040_BladeStopEoS,
	                                     iqUDT_BladeStopBoSInterface := #tUDT_DummyBladeStop);

	    END_REGION

	    REGION MCO

	        #sFB_MCOConveyLinxAixController_041(iUDT_AixConfig := #iqUDT_Configuration."041".MCO_M01,
	                                            iUDT_AixInputsModule := #iUDT_MotorInput040,
	                                            ii_PositionSetpoint := #iqUDT_RATPositioning040.Upper.EndPosition,
	                                            ix_24vOk := #ix_24vOk,
	                                            ix_SimulationModeActive := "DB_Memory".Simulation,
	                                            ii_MotorPositionId := 2,
	                                            ix_StartPositioning := #iqUDT_RATPositioning040.Upper.Start,
	                                            qUDT_HMIStatus => #iqUDT_WorkstationStatus."041".MCO_M01,
	                                            qx_Positioned => #iqUDT_RATPositioning040.Upper.Done,
	                                            iqUDT_AixOutputsModule := #iqUDT_MotorOutput040,
	                                            iqUDT_ConveyorInterface := #sUDT_Interface_041,
	                                            iqUDT_MCOStatistics := #iqUDT_WorkstationStatistics."041".MCO_M01);
	    END_REGION

	END_REGION

	IF #iqUDT_Configuration.GlobalConfig.LeftStationAvailable THEN

	    REGION 050

	        REGION Displacement
	            #sFB_Displacement050(#sUDT_Interface_050);
	        END_REGION

	        REGION Tracking

	            #sFB_Tracking_050(iUDT_ConveyorCommonConfiguration := #iqUDT_Configuration."050".Conveyor.Common,
	                              iqa_TrackingData := #sa_TrackingArray_050,
	                              iqUDT_ConveyorInterface := #sUDT_Interface_050,
	                              iqUDT_HandshakeUp := #sUDT_Handshake_040,
	                              iqUDT_Handshake := #sUDT_Handshake_050);

	        END_REGION

	        REGION EoS

	            #sFB_PECUpdate_050(iUDT_PECUpdateConfiguration := #iqUDT_Configuration."050".PEC_EoS,
	                               iUDT_ConveyorCommonConfiguration := #iqUDT_Configuration."050".Conveyor.Common,
	                               ix_PEC := NOT #iUDT_MotorInput050.AllSensorPortInputs.LeftSensor,
	                               ix_TeachingMode := FALSE,
	                               qUDT_Status => #iqUDT_WorkstationStatus."050".PEC_EoS,
	                               iqUDT_ConveyorInterface := #sUDT_Interface_050,
	                               iqUDT_UnknownGINRange := #iqUDT_UnknownGINRange,
	                               iqUDT_FifoHeader := "DB_FIFOLostGIN".Header,
	                               iqUDT_Statistics := #iqUDT_WorkstationStatistics."050".PEC_EoS,
	                               iqa_TrackingData := #sa_TrackingArray_050,
	                               iqa_FifoData := "DB_FIFOLostGIN".Data);

	        END_REGION

	        REGION Conveyor

	            //#sUDT_Handshake_050.RTR := TRUE;

	            #sUDT_Handshake_050.RTR := (#iqUDT_WorkstationStatus."060".PEC_EoS.PEC AND #sUDT_Interface_060.ActualSpeed <> 0)
	            OR (#iqUDT_WorkstationStatus."050".PEC_EoS.PEC);

	            #sFB_Conveyor_050(iUDT_ConveyorConfiguration := #iqUDT_Configuration."050".Conveyor,
	                              idi_PECEoSDistance := #iqUDT_Configuration."050".PEC_EoS.Distance,
	                              idi_PECBoSDistance := 0,
	                              ii_ExternalSpeed := 0,
	                              ix_SafetyOk := #ix_SafetyOk,
	                              ix_24vOk := #ix_24vOk,
	                              ix_400vOk := #ix_400vOk,
	                              ix_HardwareOk := TRUE,
	                              ix_PECEoS := #iqUDT_WorkstationStatus."050".PEC_EoS.PEC,
	                              ix_PECBoS := TRUE,
	                              ix_ReverseDirection := FALSE,
	                              ix_ExternalRequestDieBack := FALSE,
	                              ix_ExternalRequestHold := #sx_ReleaseBinHoldLeft,//NOT #tx_Enable,
	                              ix_ResetEnergySave := FALSE,
	                              qUDT_HMIStatus => #iqUDT_WorkstationStatus."050".Conveyor,
	                              qUDT_Status => #iqUDT_WorkstationCommonStatus."050",
	                              iqUDT_EquipmentControl := #iqUDT_EquipmentControl,
	                              iqUDT_ConveyorCommand := #iqUDT_WorkstationCommands."050".Conveyor,
	                              iqUDT_ConveyorInterface := #sUDT_Interface_050,
	                              iqUDT_HandShakeUp := #sUDT_Handshake_040,
	                              iqUDT_HandShake := #sUDT_Handshake_050,
	                              iqUDT_Statistics := #iqUDT_WorkstationStatistics."050".Conveyor);

	        END_REGION

	        REGION MCO

	            #sFB_MCOConveyLinxAixController_050(iUDT_AixConfig := #iqUDT_Configuration."050".MCO_M01,
	                                                iUDT_AixInputsModule := #iUDT_MotorInput050,
	                                                ix_24vOk := #ix_24vOk,
	                                                ix_SimulationModeActive := "DB_Memory".Simulation,
	                                                ii_MotorPositionId := 1,
	                                                qUDT_HMIStatus => #iqUDT_WorkstationStatus."050".MCO_M01,
	                                                iqUDT_AixOutputsModule := #iqUDT_MotorOutput050,
	                                                iqUDT_ConveyorInterface := #sUDT_Interface_050,
	                                                iqUDT_MCOStatistics := #iqUDT_WorkstationStatistics."050".MCO_M01);
	        END_REGION

	    END_REGION

	    REGION 060

	        REGION Displacement
	            #sFB_Displacement060(#sUDT_Interface_060);
	        END_REGION

	        REGION Tracking

	            #sFB_Tracking_060(iUDT_ConveyorCommonConfiguration := #iqUDT_Configuration."060".Conveyor.Common,
	                              iqa_TrackingData := #sa_TrackingArray_060,
	                              iqUDT_ConveyorInterface := #sUDT_Interface_060,
	                              iqUDT_HandshakeUp := #sUDT_Handshake_050,
	                              iqUDT_Handshake := #sUDT_Handshake_060);

	        END_REGION

	        REGION EoS

	            #sFB_PECUpdate_060(iUDT_PECUpdateConfiguration := #iqUDT_Configuration."060".PEC_EoS,
	                               iUDT_ConveyorCommonConfiguration := #iqUDT_Configuration."060".Conveyor.Common,
	                               ix_PEC := NOT #iUDT_MotorInput050.AllSensorPortInputs.RightSensor,
	                               ix_TeachingMode := FALSE,
	                               qUDT_Status => #iqUDT_WorkstationStatus."060".PEC_EoS,
	                               iqUDT_ConveyorInterface := #sUDT_Interface_060,
	                               iqUDT_UnknownGINRange := #iqUDT_UnknownGINRange,
	                               iqUDT_FifoHeader := "DB_FIFOLostGIN".Header,
	                               iqUDT_Statistics := #iqUDT_WorkstationStatistics."060".PEC_EoS,
	                               iqa_TrackingData := #sa_TrackingArray_060,
	                               iqa_FifoData := "DB_FIFOLostGIN".Data);

	        END_REGION

	        REGION Conveyor

	            // #sUDT_Handshake_060.RTR := TRUE;

	            #sUDT_Handshake_060.RTR := (#iqUDT_WorkstationStatus."070".PEC_EoS.PEC AND #sUDT_Interface_070.ActualSpeed <> 0)
	            OR (#iqUDT_WorkstationStatus."060".PEC_EoS.PEC);

	            #sFB_Conveyor_060(iUDT_ConveyorConfiguration := #iqUDT_Configuration."060".Conveyor,
	                              idi_PECEoSDistance := #iqUDT_Configuration."060".PEC_EoS.Distance,
	                              idi_PECBoSDistance := 0,
	                              ii_ExternalSpeed := 0,
	                              ix_SafetyOk := #ix_SafetyOk,
	                              ix_24vOk := #ix_24vOk,
	                              ix_400vOk := #ix_400vOk,
	                              ix_HardwareOk := TRUE,
	                              ix_PECEoS := #iqUDT_WorkstationStatus."060".PEC_EoS.PEC,
	                              ix_PECBoS := TRUE,
	                              ix_ReverseDirection := FALSE,
	                              ix_ExternalRequestDieBack := FALSE,
	                              ix_ExternalRequestHold := #sx_ReleaseBinHoldLeft,//NOT #tx_Enable,//(NOT #iqUDT_WorkstationStatus."035"."036".PEC_EoS.PEC AND NOT #iqUDT_WorkstationStatus."030"."031".PEC_EoS.PEC) OR (#sUDT_Interface_036.ActualSpeed = 0 AND #iqUDT_WorkstationStatus."030"."031".PEC_EoS.PEC),
	                              ix_ResetEnergySave := FALSE,
	                              qUDT_HMIStatus => #iqUDT_WorkstationStatus."060".Conveyor,
	                              qUDT_Status => #iqUDT_WorkstationCommonStatus."060",
	                              iqUDT_EquipmentControl := #iqUDT_EquipmentControl,
	                              iqUDT_ConveyorCommand := #iqUDT_WorkstationCommands."060".Conveyor,
	                              iqUDT_ConveyorInterface := #sUDT_Interface_060,
	                              iqUDT_HandShakeUp := #sUDT_Handshake_050,
	                              iqUDT_HandShake := #sUDT_Handshake_060,
	                              iqUDT_Statistics := #iqUDT_WorkstationStatistics."060".Conveyor);

	        END_REGION

	        REGION MCO

	            #sFB_MCOConveyLinxAixController_060(iUDT_AixConfig := #iqUDT_Configuration."060".MCO_M01,
	                                                iUDT_AixInputsModule := #iUDT_MotorInput050,
	                                                ix_24vOk := #ix_24vOk,
	                                                ix_SimulationModeActive := "DB_Memory".Simulation,
	                                                ii_MotorPositionId := 2,
	                                                qUDT_HMIStatus => #iqUDT_WorkstationStatus."060".MCO_M01,
	                                                iqUDT_AixOutputsModule := #iqUDT_MotorOutput050,
	                                                iqUDT_ConveyorInterface := #sUDT_Interface_060,
	                                                iqUDT_MCOStatistics := #iqUDT_WorkstationStatistics."060".MCO_M01);
	        END_REGION

	    END_REGION

	    REGION 070

	        REGION Displacement
	            #sFB_Displacement070(#sUDT_Interface_070);
	        END_REGION

	        REGION Tracking

	            #sFB_Tracking_070(iUDT_ConveyorCommonConfiguration := #iqUDT_Configuration."070".Conveyor.Common,
	                              iqa_TrackingData := #sa_TrackingArray_070,
	                              iqUDT_ConveyorInterface := #sUDT_Interface_070,
	                              iqUDT_HandshakeUp := #sUDT_Handshake_060,
	                              iqUDT_Handshake := #sUDT_Handshake_070);

	        END_REGION

	        REGION EoS

	            #sFB_PECUpdate_070(iUDT_PECUpdateConfiguration := #iqUDT_Configuration."070".PEC_EoS,
	                               iUDT_ConveyorCommonConfiguration := #iqUDT_Configuration."070".Conveyor.Common,
	                               ix_PEC := NOT #iUDT_MotorInput070.AllSensorPortInputs.LeftSensor,
	                               ix_TeachingMode := FALSE,
	                               qUDT_Status => #iqUDT_WorkstationStatus."070".PEC_EoS,
	                               iqUDT_ConveyorInterface := #sUDT_Interface_070,
	                               iqUDT_UnknownGINRange := #iqUDT_UnknownGINRange,
	                               iqUDT_FifoHeader := "DB_FIFOLostGIN".Header,
	                               iqUDT_Statistics := #iqUDT_WorkstationStatistics."070".PEC_EoS,
	                               iqa_TrackingData := #sa_TrackingArray_070,
	                               iqa_FifoData := "DB_FIFOLostGIN".Data);

	        END_REGION

	        REGION Conveyor

	            #sUDT_Handshake_070.RTR := #iqUDT_WorkstationStatus."070".PEC_EoS.PEC;

	            #sFB_Conveyor_070(iUDT_ConveyorConfiguration := #iqUDT_Configuration."070".Conveyor,
	                              idi_PECEoSDistance := #iqUDT_Configuration."070".PEC_EoS.Distance,
	                              idi_PECBoSDistance := 0,
	                              ii_ExternalSpeed := 0,
	                              ix_SafetyOk := #ix_SafetyOk,
	                              ix_24vOk := #ix_24vOk,
	                              ix_400vOk := #ix_400vOk,
	                              ix_HardwareOk := TRUE,
	                              ix_PECEoS := #iqUDT_WorkstationStatus."070".PEC_EoS.PEC,
	                              ix_PECBoS := TRUE,
	                              ix_ReverseDirection := FALSE,
	                              ix_ExternalRequestDieBack := FALSE,
	                              ix_ExternalRequestHold := #sx_ReleaseBinHoldLeft,
	                              ix_ResetEnergySave := FALSE,
	                              qUDT_HMIStatus => #iqUDT_WorkstationStatus."070".Conveyor,
	                              qUDT_Status => #iqUDT_WorkstationCommonStatus."070",
	                              iqUDT_EquipmentControl := #iqUDT_EquipmentControl,
	                              iqUDT_ConveyorCommand := #iqUDT_WorkstationCommands."070".Conveyor,
	                              iqUDT_ConveyorInterface := #sUDT_Interface_070,
	                              iqUDT_HandShakeUp := #sUDT_Handshake_060,
	                              iqUDT_HandShake := #sUDT_Handshake_070,
	                              iqUDT_Statistics := #iqUDT_WorkstationStatistics."070".Conveyor);

	        END_REGION

	        REGION MCO

	            #sFB_MCOConveyLinxAixController_070(iUDT_AixConfig := #iqUDT_Configuration."070".MCO_M01,
	                                                iUDT_AixInputsModule := #iUDT_MotorInput070,
	                                                ix_24vOk := #ix_24vOk,
	                                                ix_SimulationModeActive := "DB_Memory".Simulation,
	                                                ii_MotorPositionId := 1,
	                                                qUDT_HMIStatus => #iqUDT_WorkstationStatus."070".MCO_M01,
	                                                iqUDT_AixOutputsModule := #iqUDT_MotorOutput070,
	                                                iqUDT_ConveyorInterface := #sUDT_Interface_070,
	                                                iqUDT_MCOStatistics := #iqUDT_WorkstationStatistics."070".MCO_M01);
	        END_REGION

	    END_REGION

	END_IF;

	REGION 080

	    REGION Displacement
	        #sFB_Displacement080(#sUDT_Interface_080);
	    END_REGION

	    REGION Conveyor

	        #sUDT_Handshake_080.RTR := TRUE;

	        #sFB_Conveyor_080(iUDT_ConveyorConfiguration := #iqUDT_Configuration."080".Conveyor,
	                          idi_PECEoSDistance := 0,
	                          idi_PECBoSDistance := 0,
	                          ii_ExternalSpeed := 0,
	                          ix_SafetyOk := #ix_SafetyOk,
	                          ix_24vOk := #ix_24vOk,
	                          ix_400vOk := #ix_400vOk,
	                          ix_HardwareOk := TRUE,
	                          ix_PECEoS := TRUE,
	                          ix_PECBoS := TRUE,
	                          ix_ReverseDirection := FALSE,
	                          ix_ExternalRequestDieBack := FALSE,
	                          ix_ExternalRequestHold := #sx_Hold080,
	                          ix_ResetEnergySave := FALSE,
	                          qUDT_HMIStatus => #iqUDT_WorkstationStatus."080".Conveyor,
	                          qUDT_Status => #iqUDT_WorkstationCommonStatus."080",
	                          iqUDT_EquipmentControl := #iqUDT_EquipmentControl,
	                          iqUDT_ConveyorCommand := #iqUDT_WorkstationCommands."080".Conveyor,
	                          iqUDT_ConveyorInterface := #sUDT_Interface_080,
	                          iqUDT_HandShakeUp := #sUDT_HandshakeUp_080,
	                          iqUDT_HandShake := #sUDT_Handshake_080,
	                          iqUDT_Statistics := #iqUDT_WorkstationStatistics."080".Conveyor);

	    END_REGION

	    REGION MCO

	        #sFB_MCOConveyLinxAixController_080(iUDT_AixConfig := #iqUDT_Configuration."080".MCO_M01,
	                                            iUDT_AixInputsModule := #iUDT_MotorInput070,
	                                            ix_24vOk := #ix_24vOk,
	                                            ix_SimulationModeActive := "DB_Memory".Simulation,
	                                            ii_MotorPositionId := 2,
	                                            qUDT_HMIStatus => #iqUDT_WorkstationStatus."080".MCO_M01,
	                                            iqUDT_AixOutputsModule := #iqUDT_MotorOutput070,
	                                            iqUDT_ConveyorInterface := #sUDT_Interface_080,
	                                            iqUDT_MCOStatistics := #iqUDT_WorkstationStatistics."080".MCO_M01);
	    END_REGION

	END_REGION

	REGION 110

	    REGION Change GIN range

	        #sR_TRIG_NewParcel110(CLK := #iqUDT_HandshakeUpstream110.GIN <> 0);

	        IF #sR_TRIG_NewParcel110.Q THEN

	            #si_LastGIN110 += 1;

	            IF #si_LastGIN110 < ((#iqUDT_Configuration.GlobalConfig.GINRangeStart + #iqUDT_Configuration.GlobalConfig.GINRangeEnd) / 2) + 1
	                OR #si_LastGIN110 > #iqUDT_Configuration.GlobalConfig.GINRangeEnd
	            THEN
	                #si_LastGIN110 := ((#iqUDT_Configuration.GlobalConfig.GINRangeStart + #iqUDT_Configuration.GlobalConfig.GINRangeEnd) / 2) + 1;
	            END_IF;
	            #ts_Barcode := "DB_GIN".GIN[#iqUDT_HandshakeUpstream110.GIN].WES.Barcode;
	            #iqUDT_HandshakeUpstream110.GIN := #si_LastGIN110;

	            "DB_GIN".GIN[#iqUDT_HandshakeUpstream110.GIN] := "DB_GINDefault".GIN[#iqUDT_Configuration."110".PEC_EoS.DefaultGIN];
	            "DB_GIN".GIN[#iqUDT_HandshakeUpstream110.GIN].WES.Barcode := #ts_Barcode;

	        END_IF;

	    END_REGION

	    REGION Displacement
	        #sFB_Displacement110(#sUDT_Interface_110);
	    END_REGION

	    REGION Tracking

	        #sFB_Tracking_110(iUDT_ConveyorCommonConfiguration := #iqUDT_Configuration."110".Conveyor.Common,
	                          iqa_TrackingData := #sa_TrackingArray_110,
	                          iqUDT_ConveyorInterface := #sUDT_Interface_110,
	                          iqUDT_HandshakeUp := #iqUDT_HandshakeUpstream110,
	                          iqUDT_Handshake := #sUDT_Handshake_110);

	    END_REGION

	    REGION EoS

	        #sFB_PECUpdate_110(iUDT_PECUpdateConfiguration := #iqUDT_Configuration."110".PEC_EoS,
	                           iUDT_ConveyorCommonConfiguration := #iqUDT_Configuration."110".Conveyor.Common,
	                           ix_PEC := #iUDT_MotorInput110.AllSensorPortInputs.LeftSensor,
	                           ix_TeachingMode := FALSE,
	                           qUDT_Status => #iqUDT_WorkstationStatus."110".PEC_EoS,
	                           iqUDT_ConveyorInterface := #sUDT_Interface_110,
	                           iqUDT_UnknownGINRange := #iqUDT_UnknownGINRange,
	                           iqUDT_FifoHeader := "DB_FIFOLostGIN".Header_3,
	                           iqUDT_Statistics := #iqUDT_WorkstationStatistics."110".PEC_EoS,
	                           iqa_TrackingData := #sa_TrackingArray_110,
	                           iqa_FifoData := "DB_FIFOLostGIN".Data_3);

	    END_REGION

	    REGION Conveyor

	        #sFB_Conveyor_110(iUDT_ConveyorConfiguration := #iqUDT_Configuration."110".Conveyor,
	                          idi_PECEoSDistance := #iqUDT_Configuration."110".PEC_EoS.Distance,
	                          idi_PECBoSDistance := 0,
	                          ii_ExternalSpeed := 0,
	                          ix_SafetyOk := #ix_SafetyOk,
	                          ix_24vOk := #ix_24vOk,
	                          ix_400vOk := #ix_400vOk,
	                          ix_HardwareOk := TRUE,
	                          ix_PECEoS := #iqUDT_WorkstationStatus."110".PEC_EoS.PEC,
	                          ix_PECBoS := TRUE,
	                          ix_ReverseDirection := FALSE,
	                          ix_ExternalRequestDieBack := (#sUDT_Interface_120.ActualSpeed = 0 AND NOT #iqUDT_WorkstationStatus."110".PEC_EoS.PEC),
	                          ix_ExternalRequestHold := FALSE,
	                          ix_ResetEnergySave := FALSE,
	                          qUDT_HMIStatus => #iqUDT_WorkstationStatus."110".Conveyor,
	                          qUDT_Status => #iqUDT_WorkstationCommonStatus."110",
	                          iqUDT_EquipmentControl := #iqUDT_EquipmentControl,
	                          iqUDT_ConveyorCommand := #iqUDT_WorkstationCommands."110".Conveyor,
	                          iqUDT_ConveyorInterface := #sUDT_Interface_110,
	                          iqUDT_HandShakeUp := #iqUDT_HandshakeUpstream110,
	                          iqUDT_HandShake := #sUDT_Handshake_110,
	                          iqUDT_Statistics := #iqUDT_WorkstationStatistics."110".Conveyor);

	        //  #iqUDT_HandshakeUpstream110.RTR := #iqUDT_HandshakeUpstream110.RTR AND #iqUDT_WorkstationStatus."110".PEC_EoS.PEC;


	    END_REGION

	    REGION MCO

	        #sFB_MCOConveyLinxAixController_110(iUDT_AixConfig := #iqUDT_Configuration."110".MCO_M01,
	                                            iUDT_AixInputsModule := #iUDT_MotorInput110,
	                                            ix_24vOk := #ix_24vOk,
	                                            ix_SimulationModeActive := "DB_Memory".Simulation,
	                                            ii_MotorPositionId := 1,
	                                            qUDT_HMIStatus => #iqUDT_WorkstationStatus."110".MCO_M01,
	                                            iqUDT_AixOutputsModule := #iqUDT_MotorOutput110,
	                                            iqUDT_ConveyorInterface := #sUDT_Interface_110,
	                                            iqUDT_MCOStatistics := #iqUDT_WorkstationStatistics."110".MCO_M01);
	    END_REGION

	END_REGION

	REGION 120

	    REGION Displacement
	        #sFB_Displacement120(#sUDT_Interface_120);
	    END_REGION

	    REGION Tracking

	        #sFB_Tracking_120(iUDT_ConveyorCommonConfiguration := #iqUDT_Configuration."120".Conveyor.Common,
	                          iqa_TrackingData := #sa_TrackingArray_120,
	                          iqUDT_ConveyorInterface := #sUDT_Interface_120,
	                          iqUDT_HandshakeUp := #sUDT_Handshake_110,
	                          iqUDT_Handshake := #sUDT_Handshake_120);

	    END_REGION

	    REGION EoS

	        #sFB_PECUpdate_120(iUDT_PECUpdateConfiguration := #iqUDT_Configuration."120".PEC_EoS,
	                           iUDT_ConveyorCommonConfiguration := #iqUDT_Configuration."120".Conveyor.Common,
	                           ix_PEC := #iUDT_MotorInput110.AllSensorPortInputs.RightSensor,
	                           ix_TeachingMode := FALSE,
	                           qUDT_Status => #iqUDT_WorkstationStatus."120".PEC_EoS,
	                           iqUDT_ConveyorInterface := #sUDT_Interface_120,
	                           iqUDT_UnknownGINRange := #iqUDT_UnknownGINRange,
	                           iqUDT_FifoHeader := "DB_FIFOLostGIN".Header_1,
	                           iqUDT_Statistics := #iqUDT_WorkstationStatistics."120".PEC_EoS,
	                           iqa_TrackingData := #sa_TrackingArray_120,
	                           iqa_FifoData := "DB_FIFOLostGIN".Data_1);

	    END_REGION

	    REGION Conveyor

	        #sFB_Conveyor_120(iUDT_ConveyorConfiguration := #iqUDT_Configuration."120".Conveyor,
	                          idi_PECEoSDistance := #iqUDT_Configuration."120".PEC_EoS.Distance,
	                          idi_PECBoSDistance := 0,
	                          ii_ExternalSpeed := 0,
	                          ix_SafetyOk := #ix_SafetyOk,
	                          ix_24vOk := #ix_24vOk,
	                          ix_400vOk := #ix_400vOk,
	                          ix_HardwareOk := TRUE,
	                          ix_PECEoS := #iqUDT_WorkstationStatus."120".PEC_EoS.PEC,
	                          ix_PECBoS := TRUE,
	                          ix_ReverseDirection := FALSE,
	                          ix_ExternalRequestDieBack := #sx_Hold120 OR (#sUDT_Interface_130.ActualSpeed = 0 AND NOT #iqUDT_WorkstationStatus."120".PEC_EoS.PEC),
	                          ix_ExternalRequestHold := FALSE,
	                          ix_ResetEnergySave := FALSE,
	                          qUDT_HMIStatus => #iqUDT_WorkstationStatus."120".Conveyor,
	                          qUDT_Status => #iqUDT_WorkstationCommonStatus."120",
	                          iqUDT_EquipmentControl := #iqUDT_EquipmentControl,
	                          iqUDT_ConveyorCommand := #iqUDT_WorkstationCommands."120".Conveyor,
	                          iqUDT_ConveyorInterface := #sUDT_Interface_120,
	                          iqUDT_HandShakeUp := #sUDT_Handshake_110,
	                          iqUDT_HandShake := #sUDT_Handshake_120,
	                          iqUDT_Statistics := #iqUDT_WorkstationStatistics."120".Conveyor);

	    END_REGION

	    REGION MCO

	        #sFB_MCOConveyLinxAixController_120(iUDT_AixConfig := #iqUDT_Configuration."120".MCO_M01,
	                                            iUDT_AixInputsModule := #iUDT_MotorInput110,
	                                            ix_24vOk := #ix_24vOk,
	                                            ix_SimulationModeActive := "DB_Memory".Simulation,
	                                            ii_MotorPositionId := 2,
	                                            qUDT_HMIStatus => #iqUDT_WorkstationStatus."120".MCO_M01,
	                                            iqUDT_AixOutputsModule := #iqUDT_MotorOutput110,
	                                            iqUDT_ConveyorInterface := #sUDT_Interface_120,
	                                            iqUDT_MCOStatistics := #iqUDT_WorkstationStatistics."120".MCO_M01);
	    END_REGION

	END_REGION

	REGION 130

	    REGION Displacement
	        #sFB_Displacement130(#sUDT_Interface_130);
	    END_REGION

	    REGION Tracking

	        #sFB_Tracking_130(iUDT_ConveyorCommonConfiguration := #iqUDT_Configuration."130".Conveyor.Common,
	                          iqa_TrackingData := #sa_TrackingArray_130,
	                          iqUDT_ConveyorInterface := #sUDT_Interface_130,
	                          iqUDT_HandshakeUp := #sUDT_Handshake_120,
	                          iqUDT_Handshake := #sUDT_Handshake_130);

	    END_REGION

	    REGION EoS

	        #sFB_PECUpdate_130(iUDT_PECUpdateConfiguration := #iqUDT_Configuration."130".PEC_EoS,
	                           iUDT_ConveyorCommonConfiguration := #iqUDT_Configuration."130".Conveyor.Common,
	                           ix_PEC := #iUDT_MotorInput130.AllSensorPortInputs.LeftSensor,
	                           ix_TeachingMode := FALSE,
	                           qUDT_Status => #iqUDT_WorkstationStatus."130".PEC_EoS,
	                           iqUDT_ConveyorInterface := #sUDT_Interface_130,
	                           iqUDT_UnknownGINRange := #iqUDT_UnknownGINRange,
	                           iqUDT_FifoHeader := "DB_FIFOLostGIN".Header_2,
	                           iqUDT_Statistics := #iqUDT_WorkstationStatistics."130".PEC_EoS,
	                           iqa_TrackingData := #sa_TrackingArray_130,
	                           iqa_FifoData := "DB_FIFOLostGIN".Data_2);

	    END_REGION

	    REGION Conveyor

	        #sUDT_Handshake_130.RTR := #sUDT_Handshake_130.RTR AND NOT #sx_Hold130 OR #iqUDT_WorkstationStatus."130".PEC_EoS.PEC;

	        #sFB_Conveyor_130(iUDT_ConveyorConfiguration := #iqUDT_Configuration."130".Conveyor,
	                          idi_PECEoSDistance := #iqUDT_Configuration."130".PEC_EoS.Distance,
	                          idi_PECBoSDistance := 0,
	                          ii_ExternalSpeed := 0,
	                          ix_SafetyOk := #ix_SafetyOk,
	                          ix_24vOk := #ix_24vOk,
	                          ix_400vOk := #ix_400vOk,
	                          ix_HardwareOk := TRUE,
	                          ix_PECEoS := #iqUDT_WorkstationStatus."130".PEC_EoS.PEC,
	                          ix_PECBoS := TRUE,
	                          ix_ReverseDirection := FALSE,
	                          ix_ExternalRequestDieBack := FALSE,
	                          ix_ExternalRequestHold := #sx_Hold130,
	                          ix_ResetEnergySave := FALSE,
	                          qUDT_HMIStatus => #iqUDT_WorkstationStatus."130".Conveyor,
	                          qUDT_Status => #iqUDT_WorkstationCommonStatus."130",
	                          iqUDT_EquipmentControl := #iqUDT_EquipmentControl,
	                          iqUDT_ConveyorCommand := #iqUDT_WorkstationCommands."130".Conveyor,
	                          iqUDT_ConveyorInterface := #sUDT_Interface_130,
	                          iqUDT_HandShakeUp := #sUDT_Handshake_120,
	                          iqUDT_HandShake := #sUDT_Handshake_130,
	                          iqUDT_Statistics := #iqUDT_WorkstationStatistics."130".Conveyor);


	    END_REGION

	    REGION MCO

	        #sFB_MCOConveyLinxAixController_130(iUDT_AixConfig := #iqUDT_Configuration."130".MCO_M01,
	                                            iUDT_AixInputsModule := #iUDT_MotorInput130,
	                                            ix_24vOk := #ix_24vOk,
	                                            ix_SimulationModeActive := "DB_Memory".Simulation,
	                                            ii_MotorPositionId := 1,
	                                            qUDT_HMIStatus => #iqUDT_WorkstationStatus."130".MCO_M01,
	                                            iqUDT_AixOutputsModule := #iqUDT_MotorOutput130,
	                                            iqUDT_ConveyorInterface := #sUDT_Interface_130,
	                                            iqUDT_MCOStatistics := #iqUDT_WorkstationStatistics."130".MCO_M01);
	    END_REGION

	END_REGION

	REGION 140

	    REGION Displacement
	        #sFB_Displacement140(#sUDT_Interface_140);
	    END_REGION

	    REGION MCO

	        #sFB_MCOConveyLinxAixController_140(iUDT_AixConfig := #iqUDT_Configuration."140".MCO_M01,
	                                            iUDT_AixInputsModule := #iUDT_MotorInput140,
	                                            ii_PositionSetpoint := #iqUDT_RATPositioning140.Lower.EndPosition,
	                                            ix_24vOk := #ix_24vOk,
	                                            ix_SimulationModeActive := "DB_Memory".Simulation,
	                                            ii_MotorPositionId := 1,
	                                            ix_StartPositioning := #iqUDT_RATPositioning140.Lower.Start,
	                                            ix_ResetPosition := #iqUDT_RATPositioning140.Lower.ResetPosition,
	                                            qUDT_HMIStatus => #iqUDT_WorkstationStatus."140".MCO_M01,
	                                            qx_Positioned => #iqUDT_RATPositioning140.Lower.Done,
	                                            iqUDT_AixOutputsModule := #iqUDT_MotorOutput140,
	                                            iqUDT_ConveyorInterface := #sUDT_Interface_140,
	                                            iqUDT_MCOStatistics := #iqUDT_WorkstationStatistics."140".MCO_M01);
	    END_REGION

	    REGION BladeStopEoS

	        IF #iqUDT_Configuration.GlobalConfig.RightStationAvailable THEN

	            #sFB_BladeStopEoS_140(iUDT_Configuration := #iqUDT_Configuration."140".BladeStopEoS,
	                                  ix_IsOpened := #ix_BladeStopisUp140,
	                                  ix_IsClosed := #ix_BladeStopisDown140,
	                                  ix_AirPressureOk := TRUE,
	                                  qx_Open => #qx_BladeStopControl140,
	                                  qUDT_HMIStatus => #iqUDT_WorkstationStatus."140".BladeStopEoS,
	                                  qUDT_Statistics => #iqUDT_WorkstationStatistics."140".BladeStopEoS,
	                                  iqUDT_EquipmentControl := #iqUDT_EquipmentControl,
	                                  iqUDT_HMICommand := #iqUDT_WorkstationCommands."140".BladeStopEoS,
	                                  iqUDT_Interface := #sUDT_Interface_140_BladeStopEoS);
	        END_IF;

	    END_REGION

	END_REGION

	REGION 141

	    REGION Displacement
	        #sFB_Displacement141(#sUDT_Interface_141);
	    END_REGION

	    REGION RAT

	        #iqUDT_Configuration."141".RightAngledTransfer.BladeStopEoS := #iqUDT_Configuration.GlobalConfig.RightStationAvailable;

	        #sFB_RightAngledTransfer_141(iUDT_Configuration := #iqUDT_Configuration."141".RightAngledTransfer,
	                                     iUDT_LowerConveyorConfiguration := #iqUDT_Configuration."140".Conveyor,
	                                     iUDT_UpperConveyorConfiguration := #iqUDT_Configuration."141".Conveyor,
	                                     iUDT_PECConfiguration := #iqUDT_Configuration."140".PEC_EoS,
	                                     ii_DestinationA := #si_140DestinationA,
	                                     ii_DestinationB := #si_140DestinationB,
	                                     ii_DestinationC := #si_140DestinationC,
	                                     ii_DestinationD := #si_140DestinationD,
	                                     ix_HardwareOk := TRUE,
	                                     ix_400vOk := #ix_400vOk,
	                                     ix_24vOk := #ix_24vOk,
	                                     ix_SafetyOk := #ix_SafetyOk,
	                                     ix_AirPressureOk := #ix_AirPressureOk,
	                                     ix_SectionIsDown := #ix_SectionisDown141,
	                                     ix_SectionIsUp := #ix_SectionisUp141,
	                                     ix_ConveyorAAuto := #iqUDT_WorkstationCommonStatus."130".AutoON,
	                                     ix_ConveyorBAuto := #iqUDT_WorkstationCommonStatus."150".AutoON,
	                                     ix_ConveyorCAuto := #iqUDT_WorkstationCommonStatus."241".AutoON,
	                                     ix_ConveyorDAuto := FALSE,
	                                     ix_PEC := #iUDT_MotorInput140.AllSensorPortInputs.LeftSensor,
	                                     ix_ExternalReceiveRequestA := NOT #iqUDT_WorkstationStatus."130".PEC_EoS.PEC AND #sx_Enable1X0In,
	                                     ix_ExternalReceiveRequestB := false,
	                                     ix_ExternalReceiveRequestC := #sFB_RightAngledTransfer_241.qx_ExternalSendRequestC,
	                                     ix_ExternalReceiveRequestD := false,
	                                     ix_PECInfeedA := #iqUDT_WorkstationStatus."130".PEC_EoS.PEC,
	                                     ix_PECInfeedC := #iqUDT_WorkstationStatus."240".PEC_EoS.PEC,
	                                     qUDT_HMIRATStatus => #iqUDT_WorkstationStatus."141".RightAngledTransfer,
	                                     qUDT_HMIConveyorStatus => #iqUDT_WorkstationStatus."140".Conveyor,
	                                     qUDT_HMIPECStatus => #iqUDT_WorkstationStatus."140".PEC_EoS,
	                                     qUDT_RATStatus => #iqUDT_WorkstationCommonStatus."141",
	                                     qUDT_ConveyorStatus => #iqUDT_WorkstationCommonStatus."140",
	                                     qx_PopupControl => #qx_PopupControl141,
	                                     iqUDT_EquipmentControl := #iqUDT_EquipmentControl,
	                                     iqUDT_RATCommand := #iqUDT_WorkstationCommands."141".RightAngledTransfer,
	                                     iqUDT_ConveyorCommand := #iqUDT_WorkstationCommands."140".Conveyor,
	                                     iqUDT_RATStatistics := #iqUDT_WorkstationStatistics."141".RightAngledTransfer,
	                                     iqUDT_ConveyorStatistics := #iqUDT_WorkstationStatistics."140".Conveyor,
	                                     iqUDT_PECStatistics := #iqUDT_WorkstationStatistics."140".PEC_EoS,
	                                     iqUDT_HandShakeConveyorA := #sUDT_Handshake_130,
	                                     iqUDT_HandShakeConveyorB := #sUDT_Handshake_140,
	                                     iqUDT_HandShakeConveyorC := #sUDT_Handshake_241,
	                                     iqUDT_HandShakeConveyorD := #sUDT_Handshake_141,
	                                     iqUDT_LowerConveyorInterface := #sUDT_Interface_140,
	                                     iqUDT_UpperConveyorInterface := #sUDT_Interface_141,
	                                     iqUDT_RATPositioning := #iqUDT_RATPositioning140,
	                                     iqUDT_BladeStopEoSInterface := #sUDT_Interface_140_BladeStopEoS,
	                                     iqUDT_BladeStopBoSInterface := #tUDT_DummyBladeStop);

	    END_REGION

	    REGION MCO

	        #sFB_MCOConveyLinxAixController_141(iUDT_AixConfig := #iqUDT_Configuration."141".MCO_M01,
	                                            iUDT_AixInputsModule := #iUDT_MotorInput140,
	                                            ii_PositionSetpoint := #iqUDT_RATPositioning140.Upper.EndPosition,
	                                            ix_24vOk := #ix_24vOk,
	                                            ix_SimulationModeActive := "DB_Memory".Simulation,
	                                            ii_MotorPositionId := 2,
	                                            ix_StartPositioning := #iqUDT_RATPositioning140.Upper.Start,
	                                            qUDT_HMIStatus => #iqUDT_WorkstationStatus."141".MCO_M01,
	                                            qx_Positioned => #iqUDT_RATPositioning140.Upper.Done,
	                                            iqUDT_AixOutputsModule := #iqUDT_MotorOutput140,
	                                            iqUDT_ConveyorInterface := #sUDT_Interface_141,
	                                            iqUDT_MCOStatistics := #iqUDT_WorkstationStatistics."141".MCO_M01);
	    END_REGION

	END_REGION

	IF #iqUDT_Configuration.GlobalConfig.RightStationAvailable THEN

	    REGION 150

	        REGION Displacement
	            #sFB_Displacement150(#sUDT_Interface_150);
	        END_REGION

	        REGION Tracking

	            #sFB_Tracking_150(iUDT_ConveyorCommonConfiguration := #iqUDT_Configuration."150".Conveyor.Common,
	                              iqa_TrackingData := #sa_TrackingArray_150,
	                              iqUDT_ConveyorInterface := #sUDT_Interface_150,
	                              iqUDT_HandshakeUp := #sUDT_Handshake_140,
	                              iqUDT_Handshake := #sUDT_Handshake_150);

	        END_REGION

	        REGION EoS

	            #sFB_PECUpdate_150(iUDT_PECUpdateConfiguration := #iqUDT_Configuration."150".PEC_EoS,
	                               iUDT_ConveyorCommonConfiguration := #iqUDT_Configuration."150".Conveyor.Common,
	                               ix_PEC := NOT #iUDT_MotorInput150.AllSensorPortInputs.LeftSensor,
	                               ix_TeachingMode := FALSE,
	                               qUDT_Status => #iqUDT_WorkstationStatus."150".PEC_EoS,
	                               iqUDT_ConveyorInterface := #sUDT_Interface_150,
	                               iqUDT_UnknownGINRange := #iqUDT_UnknownGINRange,
	                               iqUDT_FifoHeader := "DB_FIFOLostGIN".Header_4,
	                               iqUDT_Statistics := #iqUDT_WorkstationStatistics."150".PEC_EoS,
	                               iqa_TrackingData := #sa_TrackingArray_150,
	                               iqa_FifoData := "DB_FIFOLostGIN".Data_4);




	        END_REGION

	        REGION Conveyor

	            #sUDT_Handshake_150.RTR := true;
	            // #tx_Enable := (#iqUDT_WorkstationStatus."160".PEC_EoS.PEC AND #sUDT_Interface_160.ActualSpeed <> 0)
	            // OR (#iqUDT_WorkstationStatus."150".PEC_EoS.PEC);
	            #sUDT_Handshake_150.RTR := (#iqUDT_WorkstationStatus."160".PEC_EoS.PEC AND #sUDT_Interface_160.ActualSpeed <> 0)
	            OR (#iqUDT_WorkstationStatus."150".PEC_EoS.PEC);
	            #sFB_Conveyor_150(iUDT_ConveyorConfiguration := #iqUDT_Configuration."150".Conveyor,
	                              idi_PECEoSDistance := #iqUDT_Configuration."150".PEC_EoS.Distance,
	                              idi_PECBoSDistance := 0,
	                              ii_ExternalSpeed := 0,
	                              ix_SafetyOk := #ix_SafetyOk,
	                              ix_24vOk := #ix_24vOk,
	                              ix_400vOk := #ix_400vOk,
	                              ix_HardwareOk := TRUE,
	                              ix_PECEoS := #iqUDT_WorkstationStatus."150".PEC_EoS.PEC,
	                              ix_PECBoS := TRUE,
	                              ix_ReverseDirection := FALSE,
	                              ix_ExternalRequestDieBack := FALSE,
	                              ix_ExternalRequestHold := #sx_ReleaseBinHoldRight,//NOT #tx_Enable,
	                              ix_ResetEnergySave := FALSE,
	                              qUDT_HMIStatus => #iqUDT_WorkstationStatus."150".Conveyor,
	                              qUDT_Status => #iqUDT_WorkstationCommonStatus."150",
	                              iqUDT_EquipmentControl := #iqUDT_EquipmentControl,
	                              iqUDT_ConveyorCommand := #iqUDT_WorkstationCommands."150".Conveyor,
	                              iqUDT_ConveyorInterface := #sUDT_Interface_150,
	                              iqUDT_HandShakeUp := #sUDT_Handshake_140,
	                              iqUDT_HandShake := #sUDT_Handshake_150,
	                              iqUDT_Statistics := #iqUDT_WorkstationStatistics."150".Conveyor);

	        END_REGION

	        REGION MCO

	            #sFB_MCOConveyLinxAixController_150(iUDT_AixConfig := #iqUDT_Configuration."150".MCO_M01,
	                                                iUDT_AixInputsModule := #iUDT_MotorInput150,
	                                                ix_24vOk := #ix_24vOk,
	                                                ix_SimulationModeActive := "DB_Memory".Simulation,
	                                                ii_MotorPositionId := 1,
	                                                qUDT_HMIStatus => #iqUDT_WorkstationStatus."150".MCO_M01,
	                                                iqUDT_AixOutputsModule := #iqUDT_MotorOutput150,
	                                                iqUDT_ConveyorInterface := #sUDT_Interface_150,
	                                                iqUDT_MCOStatistics := #iqUDT_WorkstationStatistics."150".MCO_M01);
	        END_REGION

	    END_REGION

	    REGION 160

	        REGION Displacement
	            #sFB_Displacement160(#sUDT_Interface_160);
	        END_REGION

	        REGION Tracking

	            #sFB_Tracking_160(iUDT_ConveyorCommonConfiguration := #iqUDT_Configuration."160".Conveyor.Common,
	                              iqa_TrackingData := #sa_TrackingArray_160,
	                              iqUDT_ConveyorInterface := #sUDT_Interface_160,
	                              iqUDT_HandshakeUp := #sUDT_Handshake_150,
	                              iqUDT_Handshake := #sUDT_Handshake_160);

	        END_REGION

	        REGION EoS

	            #sFB_PECUpdate_160(iUDT_PECUpdateConfiguration := #iqUDT_Configuration."160".PEC_EoS,
	                               iUDT_ConveyorCommonConfiguration := #iqUDT_Configuration."160".Conveyor.Common,
	                               ix_PEC := NOT #iUDT_MotorInput150.AllSensorPortInputs.RightSensor,
	                               ix_TeachingMode := FALSE,
	                               qUDT_Status => #iqUDT_WorkstationStatus."160".PEC_EoS,
	                               iqUDT_ConveyorInterface := #sUDT_Interface_160,
	                               iqUDT_UnknownGINRange := #iqUDT_UnknownGINRange,
	                               iqUDT_FifoHeader := "DB_FIFOLostGIN".Header_5,
	                               iqUDT_Statistics := #iqUDT_WorkstationStatistics."160".PEC_EoS,
	                               iqa_TrackingData := #sa_TrackingArray_160,
	                               iqa_FifoData := "DB_FIFOLostGIN".Data_5);




	        END_REGION

	        REGION Conveyor

	            // #sUDT_Handshake_160.RTR := true;
	            // #tx_Enable := (#iqUDT_WorkstationStatus."170".PEC_EoS.PEC AND #sUDT_Interface_170.ActualSpeed <> 0)
	            //  OR (#iqUDT_WorkstationStatus."160".PEC_EoS.PEC);
	            #sUDT_Handshake_160.RTR := (#iqUDT_WorkstationStatus."170".PEC_EoS.PEC AND #sUDT_Interface_170.ActualSpeed <> 0)
	            OR (#iqUDT_WorkstationStatus."160".PEC_EoS.PEC);


	            #sFB_Conveyor_160(iUDT_ConveyorConfiguration := #iqUDT_Configuration."160".Conveyor,
	                              idi_PECEoSDistance := #iqUDT_Configuration."160".PEC_EoS.Distance,
	                              idi_PECBoSDistance := 0,
	                              ii_ExternalSpeed := 0,
	                              ix_SafetyOk := #ix_SafetyOk,
	                              ix_24vOk := #ix_24vOk,
	                              ix_400vOk := #ix_400vOk,
	                              ix_HardwareOk := TRUE,
	                              ix_PECEoS := #iqUDT_WorkstationStatus."160".PEC_EoS.PEC,
	                              ix_PECBoS := TRUE,
	                              ix_ReverseDirection := FALSE,
	                              ix_ExternalRequestDieBack := FALSE,
	                              ix_ExternalRequestHold := #sx_ReleaseBinHoldRight,//NOT #tx_Enable,//NOT #iqUDT_WorkstationStatus."160"."132".PEC_EoS.PEC AND NOT #iqUDT_WorkstationStatus."135"."136".PEC_EoS.PEC AND NOT (#sUDT_Interface_170.ActualSpeed <> 0),
	                              ix_ResetEnergySave := FALSE,
	                              qUDT_HMIStatus => #iqUDT_WorkstationStatus."160".Conveyor,
	                              qUDT_Status => #iqUDT_WorkstationCommonStatus."160",
	                              iqUDT_EquipmentControl := #iqUDT_EquipmentControl,
	                              iqUDT_ConveyorCommand := #iqUDT_WorkstationCommands."160".Conveyor,
	                              iqUDT_ConveyorInterface := #sUDT_Interface_160,
	                              iqUDT_HandShakeUp := #sUDT_Handshake_150,
	                              iqUDT_HandShake := #sUDT_Handshake_160,
	                              iqUDT_Statistics := #iqUDT_WorkstationStatistics."160".Conveyor);

	        END_REGION

	        REGION MCO

	            #sFB_MCOConveyLinxAixController_160(iUDT_AixConfig := #iqUDT_Configuration."160".MCO_M01,
	                                                iUDT_AixInputsModule := #iUDT_MotorInput150,
	                                                ix_24vOk := #ix_24vOk,
	                                                ix_SimulationModeActive := "DB_Memory".Simulation,
	                                                ii_MotorPositionId := 2,
	                                                qUDT_HMIStatus => #iqUDT_WorkstationStatus."160".MCO_M01,
	                                                iqUDT_AixOutputsModule := #iqUDT_MotorOutput150,
	                                                iqUDT_ConveyorInterface := #sUDT_Interface_160,
	                                                iqUDT_MCOStatistics := #iqUDT_WorkstationStatistics."160".MCO_M01);
	        END_REGION

	    END_REGION

	    REGION 170

	        REGION Displacement
	            #sFB_Displacement170(#sUDT_Interface_170);
	        END_REGION

	        REGION Tracking

	            #sFB_Tracking_170(iUDT_ConveyorCommonConfiguration := #iqUDT_Configuration."170".Conveyor.Common,
	                              iqa_TrackingData := #sa_TrackingArray_170,
	                              iqUDT_ConveyorInterface := #sUDT_Interface_170,
	                              iqUDT_HandshakeUp := #sUDT_Handshake_160,
	                              iqUDT_Handshake := #sUDT_Handshake_170);

	        END_REGION

	        REGION EoS

	            #sFB_PECUpdate_170(iUDT_PECUpdateConfiguration := #iqUDT_Configuration."170".PEC_EoS,
	                               iUDT_ConveyorCommonConfiguration := #iqUDT_Configuration."170".Conveyor.Common,
	                               ix_PEC := NOT #iUDT_MotorInput170.AllSensorPortInputs.RightSensor,
	                               ix_TeachingMode := FALSE,
	                               qUDT_Status => #iqUDT_WorkstationStatus."170".PEC_EoS,
	                               iqUDT_ConveyorInterface := #sUDT_Interface_170,
	                               iqUDT_UnknownGINRange := #iqUDT_UnknownGINRange,
	                               iqUDT_FifoHeader := "DB_FIFOLostGIN".Header_6,
	                               iqUDT_Statistics := #iqUDT_WorkstationStatistics."170".PEC_EoS,
	                               iqa_TrackingData := #sa_TrackingArray_170,
	                               iqa_FifoData := "DB_FIFOLostGIN".Data_6);

	        END_REGION

	        REGION Conveyor



	            #sUDT_Handshake_170.RTR := #iqUDT_WorkstationStatus."170".PEC_EoS.PEC;

	            #sFB_Conveyor_170(iUDT_ConveyorConfiguration := #iqUDT_Configuration."170".Conveyor,
	                              idi_PECEoSDistance := #iqUDT_Configuration."170".PEC_EoS.Distance,
	                              idi_PECBoSDistance := 0,
	                              ii_ExternalSpeed := 0,
	                              ix_SafetyOk := #ix_SafetyOk,
	                              ix_24vOk := #ix_24vOk,
	                              ix_400vOk := #ix_400vOk,
	                              ix_HardwareOk := TRUE,
	                              ix_PECEoS := #iqUDT_WorkstationStatus."170".PEC_EoS.PEC,
	                              ix_PECBoS := TRUE,
	                              ix_ReverseDirection := FALSE,
	                              ix_ExternalRequestDieBack := FALSE,
	                              ix_ExternalRequestHold := #sx_ReleaseBinHoldRight,
	                              ix_ResetEnergySave := FALSE,
	                              qUDT_HMIStatus => #iqUDT_WorkstationStatus."170".Conveyor,
	                              qUDT_Status => #iqUDT_WorkstationCommonStatus."170",
	                              iqUDT_EquipmentControl := #iqUDT_EquipmentControl,
	                              iqUDT_ConveyorCommand := #iqUDT_WorkstationCommands."170".Conveyor,
	                              iqUDT_ConveyorInterface := #sUDT_Interface_170,
	                              iqUDT_HandShakeUp := #sUDT_Handshake_160,
	                              iqUDT_HandShake := #sUDT_Handshake_170,
	                              iqUDT_Statistics := #iqUDT_WorkstationStatistics."170".Conveyor);

	        END_REGION

	        REGION MCO

	            #sFB_MCOConveyLinxAixController_170(iUDT_AixConfig := #iqUDT_Configuration."170".MCO_M01,
	                                                iUDT_AixInputsModule := #iUDT_MotorInput170,
	                                                ix_24vOk := #ix_24vOk,
	                                                ix_SimulationModeActive := "DB_Memory".Simulation,
	                                                ii_MotorPositionId := 1,
	                                                qUDT_HMIStatus => #iqUDT_WorkstationStatus."170".MCO_M01,
	                                                iqUDT_AixOutputsModule := #iqUDT_MotorOutput170,
	                                                iqUDT_ConveyorInterface := #sUDT_Interface_170,
	                                                iqUDT_MCOStatistics := #iqUDT_WorkstationStatistics."170".MCO_M01);
	        END_REGION
	    END_REGION

